LIN {X 0,Y 460.515,Z 491.122,A -85,B 0,C 180,E1 -7852.428,E2 -7852.428} C_VEL
LIN {X 0,Y 460.552,Z 491.116,A -85,B 0,C 180,E1 -7855.796,E2 -7855.796} C_VEL
LIN {X 0,Y 460.531,Z 491.12,A -85,B 0,C 180,E1 -7858.234,E2 -7858.234} C_VEL
LIN {X 0,Y 460.525,Z 491.123,A -85,B 0,C 180,E1 -7861.283,E2 -7861.283} C_VEL
LIN {X 0,Y 460.526,Z 491.122,A -85,B 0,C 180,E1 -7864.503,E2 -7864.503} C_VEL
LIN {X 0,Y 460.502,Z 491.122,A -85,B 0,C 180,E1 -7867.623,E2 -7867.623} C_VEL
LIN {X 0,Y 460.528,Z 491.12,A -85,B 0,C 180,E1 -7870.267,E2 -7870.267} C_VEL
LIN {X 0,Y 460.507,Z 491.124,A -85,B 0,C 180,E1 -7873.375,E2 -7873.375} C_VEL
LIN {X 0,Y 460.512,Z 491.123,A -85,B 0,C 180,E1 -7876.625,E2 -7876.625} C_VEL
LIN {X 0,Y 460.538,Z 491.117,A -85,B 0,C 180,E1 -7879.731,E2 -7879.731} C_VEL
LIN {X 0,Y 460.499,Z 491.125,A -85,B 0,C 180,E1 -7882.524,E2 -7882.524} C_VEL
LIN {X 0,Y 460.549,Z 491.116,A -85,B 0,C 180,E1 -7885.623,E2 -7885.623} C_VEL
LIN {X 0,Y 460.541,Z 491.119,A -85,B 0,C 180,E1 -7888.744,E2 -7888.744} C_VEL
LIN {X 0,Y 460.581,Z 491.112,A -85,B 0,C 180,E1 -7892.254,E2 -7892.254} C_VEL
LIN {X 0,Y 460.529,Z 491.12,A -85,B 0,C 180,E1 -7895.667,E2 -7895.667} C_VEL
LIN {X 0,Y 460.525,Z 491.121,A -85,B 0,C 180,E1 -7898.578,E2 -7898.578} C_VEL
LIN {X 0,Y 460.588,Z 491.114,A -85,B 0,C 180,E1 -7901.31,E2 -7901.31} C_VEL
LIN {X 0,Y 460.607,Z 491.108,A -85,B 0,C 180,E1 -7904.059,E2 -7904.059} C_VEL
LIN {X 0,Y 460.612,Z 491.11,A -85,B 0,C 180,E1 -7907.666,E2 -7907.666} C_VEL
LIN {X 0,Y 460.621,Z 491.108,A -85,B 0,C 180,E1 -7911.223,E2 -7911.223} C_VEL
LIN {X 0,Y 460.685,Z 491.1,A -85,B 0,C 180,E1 -7913.869,E2 -7913.869} C_VEL
LIN {X 0,Y 460.795,Z 491.086,A -85,B 0,C 180,E1 -7917.377,E2 -7917.377} C_VEL
LIN {X 0,Y 460.853,Z 491.079,A -85,B 0,C 180,E1 -7920,E2 -7920} C_VEL
LIN {X 0,Y 460.79,Z 491.09,A -85,B 0,C 180,E1 -7922.622,E2 -7922.622} C_VEL
LIN {X 0,Y 460.681,Z 491.101,A -85,B 0,C 180,E1 -7926.13,E2 -7926.13} C_VEL
LIN {X 0,Y 460.629,Z 491.11,A -85,B 0,C 180,E1 -7928.776,E2 -7928.776} C_VEL
LIN {X 0,Y 460.637,Z 491.106,A -85,B 0,C 180,E1 -7932.457,E2 -7932.457} C_VEL
LIN {X 0,Y 460.602,Z 491.111,A -85,B 0,C 180,E1 -7935.997,E2 -7935.997} C_VEL
LIN {X 0,Y 460.57,Z 491.112,A -85,B 0,C 180,E1 -7939.615,E2 -7939.615} C_VEL
LIN {X 0,Y 460.512,Z 491.123,A -85,B 0,C 180,E1 -7942.428,E2 -7942.428} C_VEL
LIN {X 0,Y 460.55,Z 491.115,A -85,B 0,C 180,E1 -7945.797,E2 -7945.797} C_VEL
LIN {X 0,Y 460.528,Z 491.122,A -85,B 0,C 180,E1 -7948.235,E2 -7948.235} C_VEL
LIN {X 0,Y 460.522,Z 491.12,A -85,B 0,C 180,E1 -7951.283,E2 -7951.283} C_VEL
LIN {X 0,Y 460.524,Z 491.121,A -85,B 0,C 180,E1 -7954.504,E2 -7954.504} C_VEL
LIN {X 0,Y 460.502,Z 491.121,A -85,B 0,C 180,E1 -7957.623,E2 -7957.623} C_VEL
LIN {X 0,Y 460.54,Z 491.121,A -85,B 0,C 180,E1 -7960.269,E2 -7960.269} C_VEL
LIN {X 0,Y 460.5,Z 491.123,A -85,B 0,C 180,E1 -7963.375,E2 -7963.375} C_VEL
LIN {X 0,Y 460.509,Z 491.118,A -85,B 0,C 180,E1 -7966.626,E2 -7966.626} C_VEL
LIN {X 0,Y 460.567,Z 491.21,A -85,B 0,C 180,E1 -7968.772,E2 -7968.772} C_VEL
LIN {X 0,Y 462.857,Z 502.692,A -85,B 0,C 180,E1 -7972.145,E2 -7972.145} C_VEL
LIN {X 0,Y 463.542,Z 507.45,A -85,B 0,C 180,E1 -7973.472,E2 -7973.472} C_VEL
LIN {X 0,Y 463.077,Z 516.53,A -85,B 0,C 180,E1 -7975.838,E2 -7975.838} C_VEL
LIN {X 0,Y 462.397,Z 530.597,A -85,B 0,C 180,E1 -7979.391,E2 -7979.391} C_VEL
LIN {X 0,Y 461.742,Z 544.673,A -85,B 0,C 180,E1 -7982.831,E2 -7982.831} C_VEL
LIN {X 0,Y 461.237,Z 558.404,A -85,B 0,C 180,E1 -7986.098,E2 -7986.098} C_VEL
LIN {X 0,Y 460.751,Z 572.777,A -85,B 0,C 180,E1 -7989.462,E2 -7989.462} C_VEL
LIN {X 0,Y 460.448,Z 586.76,A -85,B 0,C 180,E1 -7992.684,E2 -7992.684} C_VEL
LIN {X 0,Y 460.229,Z 593.953,A -85,B 0,C 180,E1 -7994.329,E2 -7994.329} C_VEL
LIN {X 0,Y 461.606,Z 608.371,A -85,B 0,C 180,E1 -7994.74,E2 -7994.74} C_VEL
LIN {X 0,Y 462.776,Z 619.695,A -85,B 0,C 180,E1 -7995.207,E2 -7995.207} C_VEL
LIN {X 0,Y 462.309,Z 631.594,A -85,B 0,C 180,E1 -7995.81,E2 -7995.81} C_VEL
LIN {X 0,Y 461.747,Z 643.169,A -85,B 0,C 180,E1 -7996.579,E2 -7996.579} C_VEL
LIN {X 0,Y 461.287,Z 654.794,A -85,B 0,C 180,E1 -7997.56,E2 -7997.56} C_VEL
LIN {X 0,Y 460.793,Z 664.432,A -85,B 0,C 180,E1 -7998.564,E2 -7998.564} C_VEL
LIN {X 0,Y 460.421,Z 673.14,A -85,B 0,C 180,E1 -7999.668,E2 -7999.668} C_VEL
LIN {X 0,Y 460.119,Z 681.62,A -85,B 0,C 180,E1 -8000.993,E2 -8000.993} C_VEL
LIN {X 0,Y 459.968,Z 688.469,A -85,B 0,C 180,E1 -8002.317,E2 -8002.317} C_VEL
LIN {X 0,Y 459.902,Z 694.757,A -85,B 0,C 180,E1 -8003.859,E2 -8003.859} C_VEL
LIN {X 0,Y 459.871,Z 698.831,A -85,B 0,C 180,E1 -8005.178,E2 -8005.178} C_VEL
LIN {X 0,Y 459.881,Z 701.832,A -85,B 0,C 180,E1 -8006.495,E2 -8006.495} C_VEL
LIN {X 0,Y 459.866,Z 703.258,A -85,B 0,C 180,E1 -8007.372,E2 -8007.372} C_VEL
LIN {X 0,Y 459.859,Z 704.259,A -85,B 0,C 180,E1 -8008.249,E2 -8008.249} C_VEL
LIN {X 0,Y 459.967,Z 705.067,A -85,B 0,C 180,E1 -8010,E2 -8010} C_VEL
LIN {X 0,Y 459.876,Z 704.13,A -85,B 0,C 180,E1 -8011.752,E2 -8011.752} C_VEL
LIN {X 0,Y 459.89,Z 703.058,A -85,B 0,C 180,E1 -8012.628,E2 -8012.628} C_VEL
LIN {X 0,Y 459.899,Z 701.567,A -85,B 0,C 180,E1 -8013.505,E2 -8013.505} C_VEL
LIN {X 0,Y 459.901,Z 698.452,A -85,B 0,C 180,E1 -8014.821,E2 -8014.821} C_VEL
LIN {X 0,Y 459.942,Z 694.259,A -85,B 0,C 180,E1 -8016.14,E2 -8016.14} C_VEL
LIN {X 0,Y 460.005,Z 687.828,A -85,B 0,C 180,E1 -8017.683,E2 -8017.683} C_VEL
LIN {X 0,Y 460.135,Z 680.836,A -85,B 0,C 180,E1 -8019.007,E2 -8019.007} C_VEL
LIN {X 0,Y 460.422,Z 672.202,A -85,B 0,C 180,E1 -8020.332,E2 -8020.332} C_VEL
LIN {X 0,Y 460.758,Z 662.35,A -85,B 0,C 180,E1 -8021.549,E2 -8021.549} C_VEL
LIN {X 0,Y 461.262,Z 652.412,A -85,B 0,C 180,E1 -8022.55,E2 -8022.55} C_VEL
LIN {X 0,Y 461.749,Z 641.834,A -85,B 0,C 180,E1 -8023.422,E2 -8023.422} C_VEL
LIN {X 0,Y 462.281,Z 630.154,A -85,B 0,C 180,E1 -8024.191,E2 -8024.191} C_VEL
LIN {X 0,Y 462.645,Z 618.154,A -85,B 0,C 180,E1 -8024.797,E2 -8024.797} C_VEL
LIN {X 0,Y 461.586,Z 608.526,A -85,B 0,C 180,E1 -8025.208,E2 -8025.208} C_VEL
LIN {X 0,Y 460.517,Z 595.101,A -85,B 0,C 180,E1 -8025.606,E2 -8025.606} C_VEL
LIN {X 0,Y 460.253,Z 591.872,A -85,B 0,C 180,E1 -8025.698,E2 -8025.698} C_VEL
LIN {X 0,Y 460.473,Z 578.368,A -85,B 0,C 180,E1 -8028.694,E2 -8028.694} C_VEL
LIN {X 0,Y 460.805,Z 562.857,A -85,B 0,C 180,E1 -8032.178,E2 -8032.178} C_VEL
LIN {X 0,Y 461.17,Z 547.892,A -85,B 0,C 180,E1 -8035.613,E2 -8035.613} C_VEL
LIN {X 0,Y 461.528,Z 534.973,A -85,B 0,C 180,E1 -8038.664,E2 -8038.664} C_VEL
LIN {X 0,Y 462.035,Z 522.031,A -85,B 0,C 180,E1 -8041.828,E2 -8041.828} C_VEL
LIN {X 0,Y 462.623,Z 508.615,A -85,B 0,C 180,E1 -8045.26,E2 -8045.26} C_VEL
LIN {X 0,Y 462.872,Z 504.269,A -85,B 0,C 180,E1 -8046.416,E2 -8046.416} C_VEL
LIN {X 0,Y 461.961,Z 498.32,A -85,B 0,C 180,E1 -8048.127,E2 -8048.127} C_VEL
LIN {X 0,Y 460.573,Z 491.117,A -85,B 0,C 180,E1 -8050.35,E2 -8050.35} C_VEL
LIN {X 0,Y 460.503,Z 491.127,A -85,B 0,C 180,E1 -8053.376,E2 -8053.376} C_VEL
LIN {X 0,Y 460.503,Z 491.127,A -85,B 0,C 180,E1 -8056.625,E2 -8056.625} C_VEL
LIN {X 0,Y 460.545,Z 491.121,A -85,B 0,C 180,E1 -8059.731,E2 -8059.731} C_VEL
LIN {X 0,Y 460.5,Z 491.127,A -85,B 0,C 180,E1 -8062.525,E2 -8062.525} C_VEL
LIN {X 0,Y 460.539,Z 491.118,A -85,B 0,C 180,E1 -8065.623,E2 -8065.623} C_VEL
LIN {X 0,Y 460.54,Z 491.119,A -85,B 0,C 180,E1 -8068.745,E2 -8068.745} C_VEL
LIN {X 0,Y 460.585,Z 491.115,A -85,B 0,C 180,E1 -8072.254,E2 -8072.254} C_VEL
LIN {X 0,Y 460.543,Z 491.119,A -85,B 0,C 180,E1 -8074.705,E2 -8074.705} C_VEL
LIN {X 0,Y 460.514,Z 491.122,A -85,B 0,C 180,E1 -8077.572,E2 -8077.572} C_VEL
LIN {X 0,Y 460.572,Z 491.115,A -85,B 0,C 180,E1 -8080.385,E2 -8080.385} C_VEL
LIN {X 0,Y 460.608,Z 491.111,A -85,B 0,C 180,E1 -8084.059,E2 -8084.059} C_VEL
LIN {X 0,Y 460.613,Z 491.109,A -85,B 0,C 180,E1 -8087.666,E2 -8087.666} C_VEL
LIN {X 0,Y 460.631,Z 491.106,A -85,B 0,C 180,E1 -8091.224,E2 -8091.224} C_VEL
LIN {X 0,Y 460.714,Z 491.098,A -85,B 0,C 180,E1 -8093.87,E2 -8093.87} C_VEL
LIN {X 0,Y 460.793,Z 491.089,A -85,B 0,C 180,E1 -8097.378,E2 -8097.378} C_VEL
LIN {X 0,Y 460.856,Z 491.08,A -85,B 0,C 180,E1 -8100,E2 -8100} C_VEL
LIN {X 0,Y 460.804,Z 491.087,A -85,B 0,C 180,E1 -8102.623,E2 -8102.623} C_VEL
LIN {X 0,Y 460.684,Z 491.099,A -85,B 0,C 180,E1 -8106.131,E2 -8106.131} C_VEL
LIN {X 0,Y 460.632,Z 491.106,A -85,B 0,C 180,E1 -8108.776,E2 -8108.776} C_VEL
LIN {X 0,Y 460.618,Z 491.111,A -85,B 0,C 180,E1 -8112.445,E2 -8112.445} C_VEL
LIN {X 0,Y 460.605,Z 491.114,A -85,B 0,C 180,E1 -8115.998,E2 -8115.998} C_VEL
LIN {X 0,Y 460.6,Z 491.118,A -85,B 0,C 180,E1 -8119.2,E2 -8119.2} C_VEL
LIN {X 0,Y 463.456,Z 501.008,A -85,B 0,C 180,E1 -8119.852,E2 -8119.852} C_VEL
LIN {X 0,Y 463.213,Z 512.77,A -85,B 0,C 180,E1 -8120.656,E2 -8120.656} C_VEL
LIN {X 0,Y 462.751,Z 523.16,A -85,B 0,C 180,E1 -8121.552,E2 -8121.552} C_VEL
LIN {X 0,Y 462.211,Z 533.805,A -85,B 0,C 180,E1 -8122.696,E2 -8122.696} C_VEL
LIN {X 0,Y 461.756,Z 542.796,A -85,B 0,C 180,E1 -8123.913,E2 -8123.913} C_VEL
LIN {X 0,Y 461.299,Z 550.763,A -85,B 0,C 180,E1 -8125.252,E2 -8125.252} C_VEL
LIN {X 0,Y 460.951,Z 557.693,A -85,B 0,C 180,E1 -8126.73,E2 -8126.73} C_VEL
LIN {X 0,Y 460.645,Z 563.061,A -85,B 0,C 180,E1 -8128.227,E2 -8128.227} C_VEL
LIN {X 0,Y 460.477,Z 566.619,A -85,B 0,C 180,E1 -8129.545,E2 -8129.545} C_VEL
LIN {X 0,Y 460.281,Z 569.813,A -85,B 0,C 180,E1 -8131.275,E2 -8131.275} C_VEL
LIN {X 0,Y 460.157,Z 571.303,A -85,B 0,C 180,E1 -8132.857,E2 -8132.857} C_VEL
LIN {X 0,Y 460.129,Z 571.523,A -85,B 0,C 180,E1 -8134.432,E2 -8134.432} C_VEL
LIN {X 0,Y 460.139,Z 570.552,A -85,B 0,C 180,E1 -8135.952,E2 -8135.952} C_VEL
LIN {X 0,Y 460.265,Z 568.06,A -85,B 0,C 180,E1 -8137.646,E2 -8137.646} C_VEL
LIN {X 0,Y 460.451,Z 564.012,A -85,B 0,C 180,E1 -8139.326,E2 -8139.326} C_VEL
LIN {X 0,Y 460.647,Z 559.848,A -85,B 0,C 180,E1 -8140.59,E2 -8140.59} C_VEL
LIN {X 0,Y 460.947,Z 553.302,A -85,B 0,C 180,E1 -8142.134,E2 -8142.134} C_VEL
LIN {X 0,Y 461.37,Z 545.39,A -85,B 0,C 180,E1 -8143.575,E2 -8143.575} C_VEL
LIN {X 0,Y 461.841,Z 536.372,A -85,B 0,C 180,E1 -8144.887,E2 -8144.887} C_VEL
LIN {X 0,Y 462.317,Z 526.16,A -85,B 0,C 180,E1 -8146.07,E2 -8146.07} C_VEL
LIN {X 0,Y 462.788,Z 514.9,A -85,B 0,C 180,E1 -8147.116,E2 -8147.116} C_VEL
LIN {X 0,Y 463.232,Z 503.54,A -85,B 0,C 180,E1 -8147.942,E2 -8147.942} C_VEL
LIN {X 0,Y 463.212,Z 500.817,A -85,B 0,C 180,E1 -8148.119,E2 -8148.119} C_VEL
LIN {X 0,Y 460.546,Z 491.136,A -85,B 0,C 180,E1 -8148.756,E2 -8148.756} C_VEL
LIN {X 0,Y 460.52,Z 491.123,A -85,B 0,C 180,E1 -8151.266,E2 -8151.266} C_VEL
LIN {X 0,Y 460.514,Z 491.121,A -85,B 0,C 180,E1 -8154.554,E2 -8154.554} C_VEL
LIN {X 0,Y 460.537,Z 491.119,A -85,B 0,C 180,E1 -8157.716,E2 -8157.716} C_VEL
LIN {X 0,Y 460.543,Z 491.117,A -85,B 0,C 180,E1 -8160.769,E2 -8160.769} C_VEL
LIN {X 0,Y 460.548,Z 491.118,A -85,B 0,C 180,E1 -8163.734,E2 -8163.734} C_VEL
LIN {X 0,Y 460.549,Z 491.116,A -85,B 0,C 180,E1 -8166.624,E2 -8166.624} C_VEL
LIN {X 0,Y 460.556,Z 491.117,A -85,B 0,C 180,E1 -8169.453,E2 -8169.453} C_VEL
LIN {X 0,Y 460.553,Z 491.116,A -85,B 0,C 180,E1 -8172.23,E2 -8172.23} C_VEL
LIN {X 0,Y 460.543,Z 491.116,A -85,B 0,C 180,E1 -8172.589,E2 -8172.589} C_VEL
LIN {X 0,Y 459.876,Z 491.204,A -85,B 0,C 180,E1 -8173.319,E2 -8173.319} C_VEL
LIN {X 0,Y 457.008,Z 491.557,A -85,B 0,C 180,E1 -8174.504,E2 -8174.504} C_VEL
LIN {X 0,Y 454.594,Z 491.86,A -85,B 0,C 180,E1 -8175.461,E2 -8175.461} C_VEL
LIN {X 0,Y 453.576,Z 491.986,A -85,B 0,C 180,E1 -8176.2,E2 -8176.2} C_VEL
LIN {X 0,Y 453.504,Z 491.995,A -85,B 0,C 180,E1 -8176.45,E2 -8176.45} C_VEL
LIN {X 0,Y 453.536,Z 491.993,A -85,B 0,C 180,E1 -8179.283,E2 -8179.283} C_VEL
LIN {X 0,Y 453.636,Z 491.979,A -85,B 0,C 180,E1 -8182.54,E2 -8182.54} C_VEL
LIN {X 0,Y 453.663,Z 491.974,A -85,B 0,C 180,E1 -8184.667,E2 -8184.667} C_VEL
LIN {X 0,Y 453.75,Z 491.965,A -85,B 0,C 180,E1 -8187.337,E2 -8187.337} C_VEL
LIN {X 0,Y 453.821,Z 491.955,A -85,B 0,C 180,E1 -8190,E2 -8190} C_VEL
LIN {X 0,Y 453.741,Z 491.965,A -85,B 0,C 180,E1 -8192.663,E2 -8192.663} C_VEL
LIN {X 0,Y 453.649,Z 491.976,A -85,B 0,C 180,E1 -8196.226,E2 -8196.226} C_VEL
LIN {X 0,Y 453.591,Z 491.986,A -85,B 0,C 180,E1 -8198.913,E2 -8198.913} C_VEL
LIN {X 0,Y 453.569,Z 491.986,A -85,B 0,C 180,E1 -8202.529,E2 -8202.529} C_VEL
LIN {X 0,Y 453.549,Z 491.989,A -85,B 0,C 180,E1 -8206.196,E2 -8206.196} C_VEL
LIN {X 0,Y 453.522,Z 491.994,A -85,B 0,C 180,E1 -8209.039,E2 -8209.039} C_VEL
LIN {X 0,Y 453.481,Z 491.999,A -85,B 0,C 180,E1 -8211.836,E2 -8211.836} C_VEL
LIN {X 0,Y 453.499,Z 491.995,A -85,B 0,C 180,E1 -8214.735,E2 -8214.735} C_VEL
LIN {X 0,Y 453.511,Z 491.994,A -85,B 0,C 180,E1 -8217.953,E2 -8217.953} C_VEL
LIN {X 0,Y 453.479,Z 491.998,A -85,B 0,C 180,E1 -8220.759,E2 -8220.759} C_VEL
LIN {X 0,Y 453.472,Z 491.999,A -85,B 0,C 180,E1 -8223.913,E2 -8223.913} C_VEL
LIN {X 0,Y 453.453,Z 492.005,A -85,B 0,C 180,E1 -8227.19,E2 -8227.19} C_VEL
LIN {X 0,Y 453.474,Z 492,A -85,B 0,C 180,E1 -8230.611,E2 -8230.611} C_VEL
LIN {X 0,Y 453.463,Z 491.998,A -85,B 0,C 180,E1 -8234.222,E2 -8234.222} C_VEL
LIN {X 0,Y 453.451,Z 492.002,A -85,B 0,C 180,E1 -8237.003,E2 -8237.003} C_VEL
LIN {X 0,Y 453.497,Z 491.996,A -85,B 0,C 180,E1 -8239.409,E2 -8239.409} C_VEL
LIN {X 0,Y 453.452,Z 492.002,A -85,B 0,C 180,E1 -8242.81,E2 -8242.81} C_VEL
LIN {X 0,Y 453.48,Z 491.996,A -85,B 0,C 180,E1 -8246.087,E2 -8246.087} C_VEL
LIN {X 0,Y 453.48,Z 491.999,A -85,B 0,C 180,E1 -8249.24,E2 -8249.24} C_VEL
LIN {X 0,Y 453.536,Z 491.989,A -85,B 0,C 180,E1 -8252.297,E2 -8252.297} C_VEL
LIN {X 0,Y 453.499,Z 491.997,A -85,B 0,C 180,E1 -8255.264,E2 -8255.264} C_VEL
LIN {X 0,Y 453.483,Z 491.997,A -85,B 0,C 180,E1 -8258.415,E2 -8258.415} C_VEL
LIN {X 0,Y 453.525,Z 491.993,A -85,B 0,C 180,E1 -8261.008,E2 -8261.008} C_VEL
LIN {X 0,Y 453.572,Z 491.984,A -85,B 0,C 180,E1 -8263.879,E2 -8263.879} C_VEL
LIN {X 0,Y 453.567,Z 491.989,A -85,B 0,C 180,E1 -8267.471,E2 -8267.471} C_VEL
LIN {X 0,Y 453.587,Z 491.985,A -85,B 0,C 180,E1 -8271.086,E2 -8271.086} C_VEL
LIN {X 0,Y 453.651,Z 491.976,A -85,B 0,C 180,E1 -8273.774,E2 -8273.774} C_VEL
LIN {X 0,Y 453.739,Z 491.965,A -85,B 0,C 180,E1 -8277.336,E2 -8277.336} C_VEL
LIN {X 0,Y 453.822,Z 491.955,A -85,B 0,C 180,E1 -8280,E2 -8280} C_VEL
LIN {X 0,Y 453.733,Z 491.969,A -85,B 0,C 180,E1 -8282.663,E2 -8282.663} C_VEL
LIN {X 0,Y 453.648,Z 491.977,A -85,B 0,C 180,E1 -8286.226,E2 -8286.226} C_VEL
LIN {X 0,Y 453.593,Z 491.985,A -85,B 0,C 180,E1 -8288.913,E2 -8288.913} C_VEL
LIN {X 0,Y 453.604,Z 491.982,A -85,B 0,C 180,E1 -8292.55,E2 -8292.55} C_VEL
LIN {X 0,Y 453.546,Z 491.991,A -85,B 0,C 180,E1 -8296.196,E2 -8296.196} C_VEL
LIN {X 0,Y 453.52,Z 491.995,A -85,B 0,C 180,E1 -8299.039,E2 -8299.039} C_VEL
LIN {X 0,Y 453.478,Z 491.998,A -85,B 0,C 180,E1 -8301.836,E2 -8301.836} C_VEL
LIN {X 0,Y 453.501,Z 491.997,A -85,B 0,C 180,E1 -8304.735,E2 -8304.735} C_VEL
LIN {X 0,Y 453.492,Z 491.996,A -85,B 0,C 180,E1 -8307.949,E2 -8307.949} C_VEL
LIN {X 0,Y 453.477,Z 492,A -85,B 0,C 180,E1 -8310.759,E2 -8310.759} C_VEL
LIN {X 0,Y 453.469,Z 491.999,A -85,B 0,C 180,E1 -8313.913,E2 -8313.913} C_VEL
LIN {X 0,Y 453.453,Z 492.001,A -85,B 0,C 180,E1 -8317.19,E2 -8317.19} C_VEL
LIN {X 0,Y 453.495,Z 491.997,A -85,B 0,C 180,E1 -8320.609,E2 -8320.609} C_VEL
LIN {X 0,Y 453.456,Z 492.001,A -85,B 0,C 180,E1 -8323.244,E2 -8323.244} C_VEL
LIN {X 0,Y 453.461,Z 491.998,A -85,B 0,C 180,E1 -8325.778,E2 -8325.778} C_VEL
LIN {X 0,Y 453.487,Z 492.004,A -85,B 0,C 180,E1 -8328.445,E2 -8328.445} C_VEL
LIN {X 0,Y 455.388,Z 501.552,A -85,B 0,C 180,E1 -8331.316,E2 -8331.316} C_VEL
LIN {X 0,Y 456.563,Z 507.989,A -85,B 0,C 180,E1 -8333.173,E2 -8333.173} C_VEL
LIN {X 0,Y 456.325,Z 514.75,A -85,B 0,C 180,E1 -8334.979,E2 -8334.979} C_VEL
LIN {X 0,Y 455.536,Z 528.839,A -85,B 0,C 180,E1 -8338.621,E2 -8338.621} C_VEL
LIN {X 0,Y 454.948,Z 539.861,A -85,B 0,C 180,E1 -8341.387,E2 -8341.387} C_VEL
LIN {X 0,Y 454.38,Z 553.898,A -85,B 0,C 180,E1 -8344.827,E2 -8344.827} C_VEL
LIN {X 0,Y 453.842,Z 567.913,A -85,B 0,C 180,E1 -8348.182,E2 -8348.182} C_VEL
LIN {X 0,Y 453.505,Z 579.893,A -85,B 0,C 180,E1 -8351.008,E2 -8351.008} C_VEL
LIN {X 0,Y 453.186,Z 593.062,A -85,B 0,C 180,E1 -8354.084,E2 -8354.084} C_VEL
LIN {X 0,Y 454.691,Z 608.653,A -85,B 0,C 180,E1 -8354.55,E2 -8354.55} C_VEL
LIN {X 0,Y 455.77,Z 621.036,A -85,B 0,C 180,E1 -8355.089,E2 -8355.089} C_VEL
LIN {X 0,Y 455.205,Z 634.072,A -85,B 0,C 180,E1 -8355.812,E2 -8355.812} C_VEL
LIN {X 0,Y 454.66,Z 644.956,A -85,B 0,C 180,E1 -8356.593,E2 -8356.593} C_VEL
LIN {X 0,Y 454.238,Z 655.045,A -85,B 0,C 180,E1 -8357.49,E2 -8357.49} C_VEL
LIN {X 0,Y 453.708,Z 665.245,A -85,B 0,C 180,E1 -8358.609,E2 -8358.609} C_VEL
LIN {X 0,Y 453.229,Z 675.123,A -85,B 0,C 180,E1 -8359.954,E2 -8359.954} C_VEL
LIN {X 0,Y 453.003,Z 683.058,A -85,B 0,C 180,E1 -8361.3,E2 -8361.3} C_VEL
LIN {X 0,Y 452.867,Z 688.468,A -85,B 0,C 180,E1 -8362.42,E2 -8362.42} C_VEL
LIN {X 0,Y 452.825,Z 693.739,A -85,B 0,C 180,E1 -8363.763,E2 -8363.763} C_VEL
LIN {X 0,Y 452.825,Z 697.82,A -85,B 0,C 180,E1 -8365.103,E2 -8365.103} C_VEL
LIN {X 0,Y 452.839,Z 700.822,A -85,B 0,C 180,E1 -8366.441,E2 -8366.441} C_VEL
LIN {X 0,Y 452.824,Z 702.247,A -85,B 0,C 180,E1 -8367.331,E2 -8367.331} C_VEL
LIN {X 0,Y 452.824,Z 703.248,A -85,B 0,C 180,E1 -8368.221,E2 -8368.221} C_VEL
LIN {X 0,Y 452.952,Z 704.052,A -85,B 0,C 180,E1 -8370,E2 -8370} C_VEL
LIN {X 0,Y 452.843,Z 703.103,A -85,B 0,C 180,E1 -8371.779,E2 -8371.779} C_VEL
LIN {X 0,Y 452.85,Z 702.026,A -85,B 0,C 180,E1 -8372.669,E2 -8372.669} C_VEL
LIN {X 0,Y 452.857,Z 700.526,A -85,B 0,C 180,E1 -8373.559,E2 -8373.559} C_VEL
LIN {X 0,Y 452.86,Z 697.4,A -85,B 0,C 180,E1 -8374.897,E2 -8374.897} C_VEL
LIN {X 0,Y 452.888,Z 693.193,A -85,B 0,C 180,E1 -8376.236,E2 -8376.236} C_VEL
LIN {X 0,Y 452.925,Z 686.743,A -85,B 0,C 180,E1 -8377.803,E2 -8377.803} C_VEL
LIN {X 0,Y 453.088,Z 679.737,A -85,B 0,C 180,E1 -8379.149,E2 -8379.149} C_VEL
LIN {X 0,Y 453.369,Z 671.082,A -85,B 0,C 180,E1 -8380.495,E2 -8380.495} C_VEL
LIN {X 0,Y 453.676,Z 662.218,A -85,B 0,C 180,E1 -8381.618,E2 -8381.618} C_VEL
LIN {X 0,Y 454.196,Z 652.578,A -85,B 0,C 180,E1 -8382.624,E2 -8382.624} C_VEL
LIN {X 0,Y 454.788,Z 640.678,A -85,B 0,C 180,E1 -8383.631,E2 -8383.631} C_VEL
LIN {X 0,Y 455.36,Z 629.001,A -85,B 0,C 180,E1 -8384.411,E2 -8384.411} C_VEL
LIN {X 0,Y 455.64,Z 618.328,A -85,B 0,C 180,E1 -8384.973,E2 -8384.973} C_VEL
LIN {X 0,Y 454.677,Z 609.071,A -85,B 0,C 180,E1 -8385.386,E2 -8385.386} C_VEL
LIN {X 0,Y 453.648,Z 595.57,A -85,B 0,C 180,E1 -8385.825,E2 -8385.825} C_VEL
LIN {X 0,Y 453.159,Z 590.712,A -85,B 0,C 180,E1 -8385.955,E2 -8385.955} C_VEL
LIN {X 0,Y 453.429,Z 577.222,A -85,B 0,C 180,E1 -8389.006,E2 -8389.006} C_VEL
LIN {X 0,Y 453.732,Z 561.811,A -85,B 0,C 180,E1 -8392.542,E2 -8392.542} C_VEL
LIN {X 0,Y 454.164,Z 547.39,A -85,B 0,C 180,E1 -8395.926,E2 -8395.926} C_VEL
LIN {X 0,Y 454.564,Z 534.06,A -85,B 0,C 180,E1 -8399.145,E2 -8399.145} C_VEL
LIN {X 0,Y 455.081,Z 521.732,A -85,B 0,C 180,E1 -8402.232,E2 -8402.232} C_VEL
LIN {X 0,Y 455.709,Z 509.384,A -85,B 0,C 180,E1 -8405.466,E2 -8405.466} C_VEL
LIN {X 0,Y 455.881,Z 504.829,A -85,B 0,C 180,E1 -8406.712,E2 -8406.712} C_VEL
LIN {X 0,Y 454.315,Z 496.021,A -85,B 0,C 180,E1 -8409.365,E2 -8409.365} C_VEL
LIN {X 0,Y 453.517,Z 491.994,A -85,B 0,C 180,E1 -8410.68,E2 -8410.68} C_VEL
LIN {X 0,Y 453.469,Z 492.003,A -85,B 0,C 180,E1 -8414.221,E2 -8414.221} C_VEL
LIN {X 0,Y 453.466,Z 492.003,A -85,B 0,C 180,E1 -8417.005,E2 -8417.005} C_VEL
LIN {X 0,Y 453.497,Z 491.999,A -85,B 0,C 180,E1 -8419.409,E2 -8419.409} C_VEL
LIN {X 0,Y 453.45,Z 492.002,A -85,B 0,C 180,E1 -8422.228,E2 -8422.228} C_VEL
LIN {X 0,Y 453.484,Z 491.998,A -85,B 0,C 180,E1 -8425.224,E2 -8425.224} C_VEL
LIN {X 0,Y 453.469,Z 491.998,A -85,B 0,C 180,E1 -8428.475,E2 -8428.475} C_VEL
LIN {X 0,Y 453.536,Z 491.991,A -85,B 0,C 180,E1 -8432.041,E2 -8432.041} C_VEL
LIN {X 0,Y 453.504,Z 491.993,A -85,B 0,C 180,E1 -8435.265,E2 -8435.265} C_VEL
LIN {X 0,Y 453.484,Z 491.998,A -85,B 0,C 180,E1 -8438.415,E2 -8438.415} C_VEL
LIN {X 0,Y 453.526,Z 491.994,A -85,B 0,C 180,E1 -8441.009,E2 -8441.009} C_VEL
LIN {X 0,Y 453.573,Z 491.988,A -85,B 0,C 180,E1 -8443.88,E2 -8443.88} C_VEL
LIN {X 0,Y 453.568,Z 491.988,A -85,B 0,C 180,E1 -8447.471,E2 -8447.471} C_VEL
LIN {X 0,Y 453.595,Z 491.983,A -85,B 0,C 180,E1 -8451.087,E2 -8451.087} C_VEL
LIN {X 0,Y 453.682,Z 491.974,A -85,B 0,C 180,E1 -8453.775,E2 -8453.775} C_VEL
LIN {X 0,Y 453.736,Z 491.968,A -85,B 0,C 180,E1 -8457.337,E2 -8457.337} C_VEL
LIN {X 0,Y 453.826,Z 491.956,A -85,B 0,C 180,E1 -8460,E2 -8460} C_VEL
LIN {X 0,Y 453.748,Z 491.966,A -85,B 0,C 180,E1 -8462.664,E2 -8462.664} C_VEL
LIN {X 0,Y 453.65,Z 491.975,A -85,B 0,C 180,E1 -8466.226,E2 -8466.226} C_VEL
LIN {X 0,Y 453.596,Z 491.982,A -85,B 0,C 180,E1 -8468.914,E2 -8468.914} C_VEL
LIN {X 0,Y 453.568,Z 491.988,A -85,B 0,C 180,E1 -8472.529,E2 -8472.529} C_VEL
LIN {X 0,Y 453.549,Z 491.992,A -85,B 0,C 180,E1 -8476.196,E2 -8476.196} C_VEL
LIN {X 0,Y 453.582,Z 491.992,A -85,B 0,C 180,E1 -8478.938,E2 -8478.938} C_VEL
LIN {X 0,Y 456.704,Z 502.758,A -85,B 0,C 180,E1 -8479.672,E2 -8479.672} C_VEL
LIN {X 0,Y 456.378,Z 514.33,A -85,B 0,C 180,E1 -8480.485,E2 -8480.485} C_VEL
LIN {X 0,Y 455.861,Z 525.491,A -85,B 0,C 180,E1 -8481.479,E2 -8481.479} C_VEL
LIN {X 0,Y 455.348,Z 535.146,A -85,B 0,C 180,E1 -8482.549,E2 -8482.549} C_VEL
LIN {X 0,Y 454.894,Z 543.44,A -85,B 0,C 180,E1 -8483.684,E2 -8483.684} C_VEL
LIN {X 0,Y 454.434,Z 550.853,A -85,B 0,C 180,E1 -8484.925,E2 -8484.925} C_VEL
LIN {X 0,Y 454.084,Z 557.705,A -85,B 0,C 180,E1 -8486.359,E2 -8486.359} C_VEL
LIN {X 0,Y 453.748,Z 562.725,A -85,B 0,C 180,E1 -8487.689,E2 -8487.689} C_VEL
LIN {X 0,Y 453.524,Z 567.102,A -85,B 0,C 180,E1 -8489.219,E2 -8489.219} C_VEL
LIN {X 0,Y 453.309,Z 570.173,A -85,B 0,C 180,E1 -8490.773,E2 -8490.773} C_VEL
LIN {X 0,Y 453.224,Z 571.546,A -85,B 0,C 180,E1 -8491.819,E2 -8491.819} C_VEL
LIN {X 0,Y 453.149,Z 572.462,A -85,B 0,C 180,E1 -8493.122,E2 -8493.122} C_VEL
LIN {X 0,Y 453.118,Z 572.475,A -85,B 0,C 180,E1 -8494.709,E2 -8494.709} C_VEL
LIN {X 0,Y 453.145,Z 571.288,A -85,B 0,C 180,E1 -8496.245,E2 -8496.245} C_VEL
LIN {X 0,Y 453.252,Z 568.974,A -85,B 0,C 180,E1 -8497.74,E2 -8497.74} C_VEL
LIN {X 0,Y 453.469,Z 564.857,A -85,B 0,C 180,E1 -8499.452,E2 -8499.452} C_VEL
LIN {X 0,Y 453.767,Z 558.988,A -85,B 0,C 180,E1 -8501.166,E2 -8501.166} C_VEL
LIN {X 0,Y 454.083,Z 552.22,A -85,B 0,C 180,E1 -8502.663,E2 -8502.663} C_VEL
LIN {X 0,Y 454.501,Z 545.332,A -85,B 0,C 180,E1 -8503.88,E2 -8503.88} C_VEL
LIN {X 0,Y 454.955,Z 536.826,A -85,B 0,C 180,E1 -8505.107,E2 -8505.107} C_VEL
LIN {X 0,Y 455.378,Z 527.828,A -85,B 0,C 180,E1 -8506.168,E2 -8506.168} C_VEL
LIN {X 0,Y 455.857,Z 517.048,A -85,B 0,C 180,E1 -8507.2,E2 -8507.2} C_VEL
LIN {X 0,Y 456.328,Z 506.14,A -85,B 0,C 180,E1 -8508.034,E2 -8508.034} C_VEL
LIN {X 0,Y 456.398,Z 502.612,A -85,B 0,C 180,E1 -8508.264,E2 -8508.264} C_VEL
LIN {X 0,Y 453.497,Z 491.997,A -85,B 0,C 180,E1 -8508.988,E2 -8508.988} C_VEL
LIN {X 0,Y 453.451,Z 492.004,A -85,B 0,C 180,E1 -8512.228,E2 -8512.228} C_VEL
LIN {X 0,Y 453.492,Z 491.997,A -85,B 0,C 180,E1 -8515.223,E2 -8515.223} C_VEL
LIN {X 0,Y 453.471,Z 491.999,A -85,B 0,C 180,E1 -8518.475,E2 -8518.475} C_VEL
LIN {X 0,Y 453.534,Z 491.99,A -85,B 0,C 180,E1 -8522.041,E2 -8522.041} C_VEL
LIN {X 0,Y 453.501,Z 491.996,A -85,B 0,C 180,E1 -8525.265,E2 -8525.265} C_VEL
LIN {X 0,Y 453.486,Z 491.996,A -85,B 0,C 180,E1 -8528.415,E2 -8528.415} C_VEL
LIN {X 0,Y 453.528,Z 491.992,A -85,B 0,C 180,E1 -8531.009,E2 -8531.009} C_VEL
LIN {X 0,Y 453.575,Z 491.985,A -85,B 0,C 180,E1 -8533.88,E2 -8533.88} C_VEL
LIN {X 0,Y 453.504,Z 491.995,A -85,B 0,C 180,E1 -8536.45,E2 -8536.45} C_VEL
LIN {X 0,Y 452.869,Z 492.077,A -85,B 0,C 180,E1 -8537.191,E2 -8537.191} C_VEL
LIN {X 0,Y 450.04,Z 492.428,A -85,B 0,C 180,E1 -8538.396,E2 -8538.396} C_VEL
LIN {X 0,Y 447.632,Z 492.73,A -85,B 0,C 180,E1 -8539.368,E2 -8539.368} C_VEL
LIN {X 0,Y 446.6,Z 492.853,A -85,B 0,C 180,E1 -8540.118,E2 -8540.118} C_VEL
LIN {X 0,Y 446.518,Z 492.863,A -85,B 0,C 180,E1 -8540.373,E2 -8540.373} C_VEL
LIN {X 0,Y 446.618,Z 492.855,A -85,B 0,C 180,E1 -8543.676,E2 -8543.676} C_VEL
LIN {X 0,Y 446.697,Z 492.844,A -85,B 0,C 180,E1 -8547.295,E2 -8547.295} C_VEL
LIN {X 0,Y 446.79,Z 492.831,A -85,B 0,C 180,E1 -8550,E2 -8550} C_VEL
LIN {X 0,Y 446.688,Z 492.844,A -85,B 0,C 180,E1 -8552.705,E2 -8552.705} C_VEL
LIN {X 0,Y 446.617,Z 492.852,A -85,B 0,C 180,E1 -8556.324,E2 -8556.324} C_VEL
LIN {X 0,Y 446.538,Z 492.865,A -85,B 0,C 180,E1 -8559.055,E2 -8559.055} C_VEL
LIN {X 0,Y 446.527,Z 492.863,A -85,B 0,C 180,E1 -8562.73,E2 -8562.73} C_VEL
LIN {X 0,Y 446.501,Z 492.867,A -85,B 0,C 180,E1 -8566.227,E2 -8566.227} C_VEL
LIN {X 0,Y 446.473,Z 492.873,A -85,B 0,C 180,E1 -8569.303,E2 -8569.303} C_VEL
LIN {X 0,Y 446.423,Z 492.877,A -85,B 0,C 180,E1 -8572.199,E2 -8572.199} C_VEL
LIN {X 0,Y 446.443,Z 492.877,A -85,B 0,C 180,E1 -8575.153,E2 -8575.153} C_VEL
LIN {X 0,Y 446.453,Z 492.873,A -85,B 0,C 180,E1 -8578.181,E2 -8578.181} C_VEL
LIN {X 0,Y 446.42,Z 492.88,A -85,B 0,C 180,E1 -8581.3,E2 -8581.3} C_VEL
LIN {X 0,Y 446.426,Z 492.878,A -85,B 0,C 180,E1 -8584.523,E2 -8584.523} C_VEL
LIN {X 0,Y 446.414,Z 492.876,A -85,B 0,C 180,E1 -8588.078,E2 -8588.078} C_VEL
LIN {X 0,Y 446.41,Z 492.881,A -85,B 0,C 180,E1 -8591.393,E2 -8591.393} C_VEL
LIN {X 0,Y 446.453,Z 492.874,A -85,B 0,C 180,E1 -8595.104,E2 -8595.104} C_VEL
LIN {X 0,Y 446.422,Z 492.877,A -85,B 0,C 180,E1 -8598.608,E2 -8598.608} C_VEL
LIN {X 0,Y 446.427,Z 492.879,A -85,B 0,C 180,E1 -8600.971,E2 -8600.971} C_VEL
LIN {X 0,Y 446.42,Z 492.877,A -85,B 0,C 180,E1 -8604.373,E2 -8604.373} C_VEL
LIN {X 0,Y 446.426,Z 492.877,A -85,B 0,C 180,E1 -8607.638,E2 -8607.638} C_VEL
LIN {X 0,Y 446.452,Z 492.874,A -85,B 0,C 180,E1 -8610.79,E2 -8610.79} C_VEL
LIN {X 0,Y 446.463,Z 492.872,A -85,B 0,C 180,E1 -8613.847,E2 -8613.847} C_VEL
LIN {X 0,Y 446.428,Z 492.877,A -85,B 0,C 180,E1 -8616.823,E2 -8616.823} C_VEL
LIN {X 0,Y 446.446,Z 492.874,A -85,B 0,C 180,E1 -8619.737,E2 -8619.737} C_VEL
LIN {X 0,Y 446.459,Z 492.872,A -85,B 0,C 180,E1 -8622.597,E2 -8622.597} C_VEL
LIN {X 0,Y 446.471,Z 492.871,A -85,B 0,C 180,E1 -8625.412,E2 -8625.412} C_VEL
LIN {X 0,Y 446.52,Z 492.865,A -85,B 0,C 180,E1 -8628.193,E2 -8628.193} C_VEL
LIN {X 0,Y 446.535,Z 492.865,A -85,B 0,C 180,E1 -8630.944,E2 -8630.944} C_VEL
LIN {X 0,Y 446.619,Z 492.852,A -85,B 0,C 180,E1 -8633.676,E2 -8633.676} C_VEL
LIN {X 0,Y 446.686,Z 492.844,A -85,B 0,C 180,E1 -8637.294,E2 -8637.294} C_VEL
LIN {X 0,Y 446.792,Z 492.83,A -85,B 0,C 180,E1 -8640,E2 -8640} C_VEL
LIN {X 0,Y 446.68,Z 492.848,A -85,B 0,C 180,E1 -8642.705,E2 -8642.705} C_VEL
LIN {X 0,Y 446.617,Z 492.852,A -85,B 0,C 180,E1 -8646.324,E2 -8646.324} C_VEL
LIN {X 0,Y 446.539,Z 492.863,A -85,B 0,C 180,E1 -8649.055,E2 -8649.055} C_VEL
LIN {X 0,Y 446.536,Z 492.864,A -85,B 0,C 180,E1 -8652.729,E2 -8652.729} C_VEL
LIN {X 0,Y 446.49,Z 492.87,A -85,B 0,C 180,E1 -8656.459,E2 -8656.459} C_VEL
LIN {X 0,Y 446.47,Z 492.87,A -85,B 0,C 180,E1 -8659.303,E2 -8659.303} C_VEL
LIN {X 0,Y 446.42,Z 492.878,A -85,B 0,C 180,E1 -8662.199,E2 -8662.199} C_VEL
LIN {X 0,Y 446.444,Z 492.875,A -85,B 0,C 180,E1 -8665.153,E2 -8665.153} C_VEL
LIN {X 0,Y 446.441,Z 492.876,A -85,B 0,C 180,E1 -8668.182,E2 -8668.182} C_VEL
LIN {X 0,Y 446.417,Z 492.877,A -85,B 0,C 180,E1 -8671.3,E2 -8671.3} C_VEL
LIN {X 0,Y 446.424,Z 492.878,A -85,B 0,C 180,E1 -8674.523,E2 -8674.523} C_VEL
LIN {X 0,Y 446.414,Z 492.876,A -85,B 0,C 180,E1 -8678.079,E2 -8678.079} C_VEL
LIN {X 0,Y 446.429,Z 492.879,A -85,B 0,C 180,E1 -8681.391,E2 -8681.391} C_VEL
LIN {X 0,Y 446.452,Z 492.87,A -85,B 0,C 180,E1 -8685.104,E2 -8685.104} C_VEL
LIN {X 0,Y 446.45,Z 493.074,A -85,B 0,C 180,E1 -8688.193,E2 -8688.193} C_VEL
LIN {X 0,Y 448.423,Z 502.801,A -85,B 0,C 180,E1 -8691.178,E2 -8691.178} C_VEL
LIN {X 0,Y 449.653,Z 509.818,A -85,B 0,C 180,E1 -8693.229,E2 -8693.229} C_VEL
LIN {X 0,Y 449.159,Z 519.04,A -85,B 0,C 180,E1 -8695.716,E2 -8695.716} C_VEL
LIN {X 0,Y 448.412,Z 532.605,A -85,B 0,C 180,E1 -8699.258,E2 -8699.258} C_VEL
LIN {X 0,Y 447.637,Z 547.054,A -85,B 0,C 180,E1 -8702.915,E2 -8702.915} C_VEL
LIN {X 0,Y 447.128,Z 559.077,A -85,B 0,C 180,E1 -8705.879,E2 -8705.879} C_VEL
LIN {X 0,Y 446.634,Z 573.009,A -85,B 0,C 180,E1 -8709.265,E2 -8709.265} C_VEL
LIN {X 0,Y 446.29,Z 586.929,A -85,B 0,C 180,E1 -8712.59,E2 -8712.59} C_VEL
LIN {X 0,Y 446.152,Z 592.452,A -85,B 0,C 180,E1 -8713.852,E2 -8713.852} C_VEL
LIN {X 0,Y 447.535,Z 606.314,A -85,B 0,C 180,E1 -8714.26,E2 -8714.26} C_VEL
LIN {X 0,Y 448.487,Z 617.342,A -85,B 0,C 180,E1 -8714.725,E2 -8714.725} C_VEL
LIN {X 0,Y 448.76,Z 622.157,A -85,B 0,C 180,E1 -8714.967,E2 -8714.967} C_VEL
LIN {X 0,Y 448.185,Z 634.73,A -85,B 0,C 180,E1 -8715.701,E2 -8715.701} C_VEL
LIN {X 0,Y 447.564,Z 646.199,A -85,B 0,C 180,E1 -8716.574,E2 -8716.574} C_VEL
LIN {X 0,Y 447.154,Z 656.18,A -85,B 0,C 180,E1 -8717.519,E2 -8717.519} C_VEL
LIN {X 0,Y 446.644,Z 664.188,A -85,B 0,C 180,E1 -8718.427,E2 -8718.427} C_VEL
LIN {X 0,Y 446.193,Z 674.08,A -85,B 0,C 180,E1 -8719.793,E2 -8719.793} C_VEL
LIN {X 0,Y 445.932,Z 682.025,A -85,B 0,C 180,E1 -8721.161,E2 -8721.161} C_VEL
LIN {X 0,Y 445.822,Z 687.442,A -85,B 0,C 180,E1 -8722.3,E2 -8722.3} C_VEL
LIN {X 0,Y 445.756,Z 692.716,A -85,B 0,C 180,E1 -8723.664,E2 -8723.664} C_VEL
LIN {X 0,Y 445.778,Z 696.805,A -85,B 0,C 180,E1 -8725.026,E2 -8725.026} C_VEL
LIN {X 0,Y 445.799,Z 699.808,A -85,B 0,C 180,E1 -8726.385,E2 -8726.385} C_VEL
LIN {X 0,Y 445.783,Z 701.235,A -85,B 0,C 180,E1 -8727.289,E2 -8727.289} C_VEL
LIN {X 0,Y 445.788,Z 702.236,A -85,B 0,C 180,E1 -8728.193,E2 -8728.193} C_VEL
LIN {X 0,Y 445.936,Z 703.036,A -85,B 0,C 180,E1 -8730,E2 -8730} C_VEL
LIN {X 0,Y 445.809,Z 702.079,A -85,B 0,C 180,E1 -8731.807,E2 -8731.807} C_VEL
LIN {X 0,Y 445.81,Z 700.991,A -85,B 0,C 180,E1 -8732.711,E2 -8732.711} C_VEL
LIN {X 0,Y 445.816,Z 699.486,A -85,B 0,C 180,E1 -8733.615,E2 -8733.615} C_VEL
LIN {X 0,Y 445.817,Z 696.349,A -85,B 0,C 180,E1 -8734.974,E2 -8734.974} C_VEL
LIN {X 0,Y 445.811,Z 692.123,A -85,B 0,C 180,E1 -8736.336,E2 -8736.336} C_VEL
LIN {X 0,Y 445.877,Z 685.66,A -85,B 0,C 180,E1 -8737.928,E2 -8737.928} C_VEL
LIN {X 0,Y 446.042,Z 678.634,A -85,B 0,C 180,E1 -8739.294,E2 -8739.294} C_VEL
LIN {X 0,Y 446.341,Z 669.965,A -85,B 0,C 180,E1 -8740.662,E2 -8740.662} C_VEL
LIN {X 0,Y 446.747,Z 660.103,A -85,B 0,C 180,E1 -8741.916,E2 -8741.916} C_VEL
LIN {X 0,Y 447.104,Z 651.607,A -85,B 0,C 180,E1 -8742.814,E2 -8742.814} C_VEL
LIN {X 0,Y 447.811,Z 639.603,A -85,B 0,C 180,E1 -8743.848,E2 -8743.848} C_VEL
LIN {X 0,Y 448.422,Z 627.976,A -85,B 0,C 180,E1 -8744.639,E2 -8744.639} C_VEL
LIN {X 0,Y 448.737,Z 619.639,A -85,B 0,C 180,E1 -8745.093,E2 -8745.093} C_VEL
LIN {X 0,Y 447.775,Z 609.911,A -85,B 0,C 180,E1 -8745.56,E2 -8745.56} C_VEL
LIN {X 0,Y 446.802,Z 596.349,A -85,B 0,C 180,E1 -8746.035,E2 -8746.035} C_VEL
LIN {X 0,Y 446.11,Z 589.547,A -85,B 0,C 180,E1 -8746.225,E2 -8746.225} C_VEL
LIN {X 0,Y 446.368,Z 576.192,A -85,B 0,C 180,E1 -8749.308,E2 -8749.308} C_VEL
LIN {X 0,Y 446.66,Z 561.81,A -85,B 0,C 180,E1 -8752.675,E2 -8752.675} C_VEL
LIN {X 0,Y 447.103,Z 548.489,A -85,B 0,C 180,E1 -8755.862,E2 -8755.862} C_VEL
LIN {X 0,Y 447.523,Z 535.194,A -85,B 0,C 180,E1 -8759.133,E2 -8759.133} C_VEL
LIN {X 0,Y 448.075,Z 523.062,A -85,B 0,C 180,E1 -8762.228,E2 -8762.228} C_VEL
LIN {X 0,Y 448.729,Z 510.927,A -85,B 0,C 180,E1 -8765.469,E2 -8765.469} C_VEL
LIN {X 0,Y 448.872,Z 505.42,A -85,B 0,C 180,E1 -8767.012,E2 -8767.012} C_VEL
LIN {X 0,Y 446.992,Z 495.407,A -85,B 0,C 180,E1 -8770.139,E2 -8770.139} C_VEL
LIN {X 0,Y 446.466,Z 492.871,A -85,B 0,C 180,E1 -8771.018,E2 -8771.018} C_VEL
LIN {X 0,Y 446.404,Z 492.885,A -85,B 0,C 180,E1 -8773.846,E2 -8773.846} C_VEL
LIN {X 0,Y 446.402,Z 492.885,A -85,B 0,C 180,E1 -8776.403,E2 -8776.403} C_VEL
LIN {X 0,Y 446.43,Z 492.879,A -85,B 0,C 180,E1 -8779.083,E2 -8779.083} C_VEL
LIN {X 0,Y 446.41,Z 492.878,A -85,B 0,C 180,E1 -8782.121,E2 -8782.121} C_VEL
LIN {X 0,Y 446.425,Z 492.876,A -85,B 0,C 180,E1 -8785.477,E2 -8785.477} C_VEL
LIN {X 0,Y 446.419,Z 492.877,A -85,B 0,C 180,E1 -8788.7,E2 -8788.7} C_VEL
LIN {X 0,Y 446.488,Z 492.868,A -85,B 0,C 180,E1 -8791.822,E2 -8791.822} C_VEL
LIN {X 0,Y 446.447,Z 492.875,A -85,B 0,C 180,E1 -8794.847,E2 -8794.847} C_VEL
LIN {X 0,Y 446.452,Z 492.873,A -85,B 0,C 180,E1 -8798.245,E2 -8798.245} C_VEL
LIN {X 0,Y 446.455,Z 492.871,A -85,B 0,C 180,E1 -8801.649,E2 -8801.649} C_VEL
LIN {X 0,Y 446.511,Z 492.867,A -85,B 0,C 180,E1 -8804.48,E2 -8804.48} C_VEL
LIN {X 0,Y 446.521,Z 492.864,A -85,B 0,C 180,E1 -8808.193,E2 -8808.193} C_VEL
LIN {X 0,Y 446.604,Z 492.852,A -85,B 0,C 180,E1 -8811.858,E2 -8811.858} C_VEL
LIN {X 0,Y 446.649,Z 492.849,A -85,B 0,C 180,E1 -8814.583,E2 -8814.583} C_VEL
LIN {X 0,Y 446.667,Z 492.847,A -85,B 0,C 180,E1 -8818.197,E2 -8818.197} C_VEL
LIN {X 0,Y 446.796,Z 492.832,A -85,B 0,C 180,E1 -8820,E2 -8820} C_VEL
LIN {X 0,Y 446.695,Z 492.845,A -85,B 0,C 180,E1 -8822.706,E2 -8822.706} C_VEL
LIN {X 0,Y 446.619,Z 492.851,A -85,B 0,C 180,E1 -8826.324,E2 -8826.324} C_VEL
LIN {X 0,Y 446.541,Z 492.861,A -85,B 0,C 180,E1 -8829.056,E2 -8829.056} C_VEL
LIN {X 0,Y 446.526,Z 492.865,A -85,B 0,C 180,E1 -8832.73,E2 -8832.73} C_VEL
LIN {X 0,Y 446.5,Z 492.87,A -85,B 0,C 180,E1 -8836.228,E2 -8836.228} C_VEL
LIN {X 0,Y 446.549,Z 493.071,A -85,B 0,C 180,E1 -8838.685,E2 -8838.685} C_VEL
LIN {X 0,Y 449.97,Z 504.803,A -85,B 0,C 180,E1 -8839.503,E2 -8839.503} C_VEL
LIN {X 0,Y 449.538,Z 516.454,A -85,B 0,C 180,E1 -8840.353,E2 -8840.353} C_VEL
LIN {X 0,Y 449.03,Z 527.174,A -85,B 0,C 180,E1 -8841.34,E2 -8841.34} C_VEL
LIN {X 0,Y 448.47,Z 536.442,A -85,B 0,C 180,E1 -8842.392,E2 -8842.392} C_VEL
LIN {X 0,Y 447.973,Z 544.929,A -85,B 0,C 180,E1 -8843.582,E2 -8843.582} C_VEL
LIN {X 0,Y 447.497,Z 552.523,A -85,B 0,C 180,E1 -8844.892,E2 -8844.892} C_VEL
LIN {X 0,Y 447.11,Z 559.339,A -85,B 0,C 180,E1 -8846.366,E2 -8846.366} C_VEL
LIN {X 0,Y 446.778,Z 564.011,A -85,B 0,C 180,E1 -8847.649,E2 -8847.649} C_VEL
LIN {X 0,Y 446.525,Z 568.311,A -85,B 0,C 180,E1 -8849.204,E2 -8849.204} C_VEL
LIN {X 0,Y 446.362,Z 570.464,A -85,B 0,C 180,E1 -8850.255,E2 -8850.255} C_VEL
LIN {X 0,Y 446.213,Z 572.538,A -85,B 0,C 180,E1 -8851.731,E2 -8851.731} C_VEL
LIN {X 0,Y 446.121,Z 573.61,A -85,B 0,C 180,E1 -8853.462,E2 -8853.462} C_VEL
LIN {X 0,Y 446.097,Z 573.355,A -85,B 0,C 180,E1 -8854.992,E2 -8854.992} C_VEL
LIN {X 0,Y 446.158,Z 571.655,A -85,B 0,C 180,E1 -8856.769,E2 -8856.769} C_VEL
LIN {X 0,Y 446.323,Z 568.481,A -85,B 0,C 180,E1 -8858.5,E2 -8858.5} C_VEL
LIN {X 0,Y 446.567,Z 563.841,A -85,B 0,C 180,E1 -8860.185,E2 -8860.185} C_VEL
LIN {X 0,Y 446.847,Z 558.623,A -85,B 0,C 180,E1 -8861.602,E2 -8861.602} C_VEL
LIN {X 0,Y 447.155,Z 552.979,A -85,B 0,C 180,E1 -8862.826,E2 -8862.826} C_VEL
LIN {X 0,Y 447.568,Z 546.317,A -85,B 0,C 180,E1 -8864.015,E2 -8864.015} C_VEL
LIN {X 0,Y 448.05,Z 537.645,A -85,B 0,C 180,E1 -8865.281,E2 -8865.281} C_VEL
LIN {X 0,Y 448.539,Z 528.073,A -85,B 0,C 180,E1 -8866.415,E2 -8866.415} C_VEL
LIN {X 0,Y 449.052,Z 516.771,A -85,B 0,C 180,E1 -8867.496,E2 -8867.496} C_VEL
LIN {X 0,Y 449.546,Z 505.169,A -85,B 0,C 180,E1 -8868.361,E2 -8868.361} C_VEL
LIN {X 0,Y 448.599,Z 500.419,A -85,B 0,C 180,E1 -8868.703,E2 -8868.703} C_VEL
LIN {X 0,Y 446.432,Z 492.878,A -85,B 0,C 180,E1 -8869.236,E2 -8869.236} C_VEL
LIN {X 0,Y 446.41,Z 492.88,A -85,B 0,C 180,E1 -8872.121,E2 -8872.121} C_VEL
LIN {X 0,Y 446.434,Z 492.878,A -85,B 0,C 180,E1 -8875.477,E2 -8875.477} C_VEL
LIN {X 0,Y 446.421,Z 492.878,A -85,B 0,C 180,E1 -8878.7,E2 -8878.7} C_VEL
LIN {X 0,Y 446.49,Z 492.868,A -85,B 0,C 180,E1 -8881.821,E2 -8881.821} C_VEL
LIN {X 0,Y 446.445,Z 492.876,A -85,B 0,C 180,E1 -8884.847,E2 -8884.847} C_VEL
LIN {X 0,Y 446.454,Z 492.872,A -85,B 0,C 180,E1 -8888.245,E2 -8888.245} C_VEL
LIN {X 0,Y 446.456,Z 492.875,A -85,B 0,C 180,E1 -8891.649,E2 -8891.649} C_VEL
LIN {X 0,Y 446.513,Z 492.864,A -85,B 0,C 180,E1 -8894.48,E2 -8894.48} C_VEL
LIN {X 0,Y 446.523,Z 492.863,A -85,B 0,C 180,E1 -8898.193,E2 -8898.193} C_VEL
LIN {X 0,Y 446.518,Z 492.863,A -85,B 0,C 180,E1 -8900.373,E2 -8900.373} C_VEL
LIN {X 0,Y 445.856,Z 492.95,A -85,B 0,C 180,E1 -8901.126,E2 -8901.126} C_VEL
LIN {X 0,Y 443.017,Z 493.301,A -85,B 0,C 180,E1 -8902.35,E2 -8902.35} C_VEL
LIN {X 0,Y 440.64,Z 493.598,A -85,B 0,C 180,E1 -8903.337,E2 -8903.337} C_VEL
LIN {X 0,Y 439.657,Z 493.719,A -85,B 0,C 180,E1 -8904.1,E2 -8904.1} C_VEL
LIN {X 0,Y 439.597,Z 493.726,A -85,B 0,C 180,E1 -8904.358,E2 -8904.358} C_VEL
LIN {X 0,Y 439.638,Z 493.722,A -85,B 0,C 180,E1 -8908.168,E2 -8908.168} C_VEL
LIN {X 0,Y 439.76,Z 493.706,A -85,B 0,C 180,E1 -8910,E2 -8910} C_VEL
LIN {X 0,Y 439.637,Z 493.722,A -85,B 0,C 180,E1 -8912.749,E2 -8912.749} C_VEL
LIN {X 0,Y 439.569,Z 493.73,A -85,B 0,C 180,E1 -8916.426,E2 -8916.426} C_VEL
LIN {X 0,Y 439.501,Z 493.741,A -85,B 0,C 180,E1 -8919.202,E2 -8919.202} C_VEL
LIN {X 0,Y 439.471,Z 493.743,A -85,B 0,C 180,E1 -8922.937,E2 -8922.937} C_VEL
LIN {X 0,Y 439.451,Z 493.745,A -85,B 0,C 180,E1 -8926.348,E2 -8926.348} C_VEL
LIN {X 0,Y 439.407,Z 493.75,A -85,B 0,C 180,E1 -8929.626,E2 -8929.626} C_VEL
LIN {X 0,Y 439.368,Z 493.757,A -85,B 0,C 180,E1 -8932.575,E2 -8932.575} C_VEL
LIN {X 0,Y 439.382,Z 493.754,A -85,B 0,C 180,E1 -8935.586,E2 -8935.586} C_VEL
LIN {X 0,Y 439.404,Z 493.753,A -85,B 0,C 180,E1 -8938.674,E2 -8938.674} C_VEL
LIN {X 0,Y 439.373,Z 493.753,A -85,B 0,C 180,E1 -8942.03,E2 -8942.03} C_VEL
LIN {X 0,Y 439.395,Z 493.754,A -85,B 0,C 180,E1 -8945.339,E2 -8945.339} C_VEL
LIN {X 0,Y 439.371,Z 493.755,A -85,B 0,C 180,E1 -8948.596,E2 -8948.596} C_VEL
LIN {X 0,Y 439.371,Z 493.757,A -85,B 0,C 180,E1 -8951.253,E2 -8951.253} C_VEL
LIN {X 0,Y 439.401,Z 493.753,A -85,B 0,C 180,E1 -8954.729,E2 -8954.729} C_VEL
LIN {X 0,Y 439.387,Z 493.753,A -85,B 0,C 180,E1 -8957.794,E2 -8957.794} C_VEL
LIN {X 0,Y 439.392,Z 493.751,A -85,B 0,C 180,E1 -8960.223,E2 -8960.223} C_VEL
LIN {X 0,Y 439.375,Z 493.755,A -85,B 0,C 180,E1 -8963.712,E2 -8963.712} C_VEL
LIN {X 0,Y 439.376,Z 493.756,A -85,B 0,C 180,E1 -8967.054,E2 -8967.054} C_VEL
LIN {X 0,Y 439.386,Z 493.753,A -85,B 0,C 180,E1 -8970.274,E2 -8970.274} C_VEL
LIN {X 0,Y 439.422,Z 493.749,A -85,B 0,C 180,E1 -8973.395,E2 -8973.395} C_VEL
LIN {X 0,Y 439.386,Z 493.753,A -85,B 0,C 180,E1 -8976.429,E2 -8976.429} C_VEL
LIN {X 0,Y 439.391,Z 493.753,A -85,B 0,C 180,E1 -8979.397,E2 -8979.397} C_VEL
LIN {X 0,Y 439.428,Z 493.748,A -85,B 0,C 180,E1 -8982.309,E2 -8982.309} C_VEL
LIN {X 0,Y 439.449,Z 493.746,A -85,B 0,C 180,E1 -8985.174,E2 -8985.174} C_VEL
LIN {X 0,Y 439.486,Z 493.74,A -85,B 0,C 180,E1 -8988.001,E2 -8988.001} C_VEL
LIN {X 0,Y 439.506,Z 493.738,A -85,B 0,C 180,E1 -8991.725,E2 -8991.725} C_VEL
LIN {X 0,Y 439.611,Z 493.725,A -85,B 0,C 180,E1 -8994.495,E2 -8994.495} C_VEL
LIN {X 0,Y 439.634,Z 493.723,A -85,B 0,C 180,E1 -8998.168,E2 -8998.168} C_VEL
LIN {X 0,Y 439.761,Z 493.706,A -85,B 0,C 180,E1 -9000,E2 -9000} C_VEL
LIN {X 0,Y 439.629,Z 493.726,A -85,B 0,C 180,E1 -9002.749,E2 -9002.749} C_VEL
LIN {X 0,Y 439.568,Z 493.73,A -85,B 0,C 180,E1 -9006.426,E2 -9006.426} C_VEL
LIN {X 0,Y 439.501,Z 493.739,A -85,B 0,C 180,E1 -9009.201,E2 -9009.201} C_VEL
LIN {X 0,Y 439.506,Z 493.74,A -85,B 0,C 180,E1 -9012.726,E2 -9012.726} C_VEL
LIN {X 0,Y 439.448,Z 493.747,A -85,B 0,C 180,E1 -9016.348,E2 -9016.348} C_VEL
LIN {X 0,Y 439.404,Z 493.749,A -85,B 0,C 180,E1 -9019.626,E2 -9019.626} C_VEL
LIN {X 0,Y 439.365,Z 493.757,A -85,B 0,C 180,E1 -9022.575,E2 -9022.575} C_VEL
LIN {X 0,Y 439.381,Z 493.752,A -85,B 0,C 180,E1 -9025.586,E2 -9025.586} C_VEL
LIN {X 0,Y 439.398,Z 493.753,A -85,B 0,C 180,E1 -9028.675,E2 -9028.675} C_VEL
LIN {X 0,Y 439.37,Z 493.753,A -85,B 0,C 180,E1 -9032.03,E2 -9032.03} C_VEL
LIN {X 0,Y 439.393,Z 493.753,A -85,B 0,C 180,E1 -9035.34,E2 -9035.34} C_VEL
LIN {X 0,Y 439.371,Z 493.758,A -85,B 0,C 180,E1 -9038.596,E2 -9038.596} C_VEL
LIN {X 0,Y 439.39,Z 493.755,A -85,B 0,C 180,E1 -9041.257,E2 -9041.257} C_VEL
LIN {X 0,Y 439.4,Z 493.75,A -85,B 0,C 180,E1 -9044.729,E2 -9044.729} C_VEL
LIN {X 0,Y 439.42,Z 493.909,A -85,B 0,C 180,E1 -9047.872,E2 -9047.872} C_VEL
LIN {X 0,Y 441.332,Z 503.542,A -85,B 0,C 180,E1 -9050.886,E2 -9050.886} C_VEL
LIN {X 0,Y 442.708,Z 511.242,A -85,B 0,C 180,E1 -9053.181,E2 -9053.181} C_VEL
LIN {X 0,Y 442.144,Z 520.61,A -85,B 0,C 180,E1 -9055.747,E2 -9055.747} C_VEL
LIN {X 0,Y 441.365,Z 534.257,A -85,B 0,C 180,E1 -9059.366,E2 -9059.366} C_VEL
LIN {X 0,Y 440.59,Z 548.095,A -85,B 0,C 180,E1 -9062.929,E2 -9062.929} C_VEL
LIN {X 0,Y 440.048,Z 560.266,A -85,B 0,C 180,E1 -9065.992,E2 -9065.992} C_VEL
LIN {X 0,Y 439.557,Z 574.092,A -85,B 0,C 180,E1 -9069.405,E2 -9069.405} C_VEL
LIN {X 0,Y 439.186,Z 587.944,A -85,B 0,C 180,E1 -9072.78,E2 -9072.78} C_VEL
LIN {X 0,Y 439.081,Z 591.313,A -85,B 0,C 180,E1 -9073.595,E2 -9073.595} C_VEL
LIN {X 0,Y 440.491,Z 605.574,A -85,B 0,C 180,E1 -9074.024,E2 -9074.024} C_VEL
LIN {X 0,Y 441.43,Z 617.372,A -85,B 0,C 180,E1 -9074.533,E2 -9074.533} C_VEL
LIN {X 0,Y 441.814,Z 622.092,A -85,B 0,C 180,E1 -9074.783,E2 -9074.783} C_VEL
LIN {X 0,Y 441.247,Z 633.596,A -85,B 0,C 180,E1 -9075.472,E2 -9075.472} C_VEL
LIN {X 0,Y 440.587,Z 645.474,A -85,B 0,C 180,E1 -9076.39,E2 -9076.39} C_VEL
LIN {X 0,Y 440.121,Z 655.111,A -85,B 0,C 180,E1 -9077.317,E2 -9077.317} C_VEL
LIN {X 0,Y 439.56,Z 664.944,A -85,B 0,C 180,E1 -9078.471,E2 -9078.471} C_VEL
LIN {X 0,Y 439.167,Z 673.038,A -85,B 0,C 180,E1 -9079.628,E2 -9079.628} C_VEL
LIN {X 0,Y 438.867,Z 680.992,A -85,B 0,C 180,E1 -9081.017,E2 -9081.017} C_VEL
LIN {X 0,Y 438.759,Z 686.413,A -85,B 0,C 180,E1 -9082.175,E2 -9082.175} C_VEL
LIN {X 0,Y 438.681,Z 691.692,A -85,B 0,C 180,E1 -9083.561,E2 -9083.561} C_VEL
LIN {X 0,Y 438.732,Z 695.788,A -85,B 0,C 180,E1 -9084.946,E2 -9084.946} C_VEL
LIN {X 0,Y 438.759,Z 698.794,A -85,B 0,C 180,E1 -9086.327,E2 -9086.327} C_VEL
LIN {X 0,Y 438.742,Z 700.222,A -85,B 0,C 180,E1 -9087.246,E2 -9087.246} C_VEL
LIN {X 0,Y 438.753,Z 701.221,A -85,B 0,C 180,E1 -9088.164,E2 -9088.164} C_VEL
LIN {X 0,Y 438.919,Z 702.019,A -85,B 0,C 180,E1 -9090,E2 -9090} C_VEL
LIN {X 0,Y 438.775,Z 701.05,A -85,B 0,C 180,E1 -9091.836,E2 -9091.836} C_VEL
LIN {X 0,Y 438.77,Z 699.957,A -85,B 0,C 180,E1 -9092.754,E2 -9092.754} C_VEL
LIN {X 0,Y 438.766,Z 697.489,A -85,B 0,C 180,E1 -9094.134,E2 -9094.134} C_VEL
LIN {X 0,Y 438.729,Z 693.981,A -85,B 0,C 180,E1 -9095.516,E2 -9095.516} C_VEL
LIN {X 0,Y 438.758,Z 688.89,A -85,B 0,C 180,E1 -9097.028,E2 -9097.028} C_VEL
LIN {X 0,Y 438.873,Z 682.433,A -85,B 0,C 180,E1 -9098.519,E2 -9098.519} C_VEL
LIN {X 0,Y 439.027,Z 674.862,A -85,B 0,C 180,E1 -9099.909,E2 -9099.909} C_VEL
LIN {X 0,Y 439.482,Z 665.544,A -85,B 0,C 180,E1 -9101.297,E2 -9101.297} C_VEL
LIN {X 0,Y 440.03,Z 656.021,A -85,B 0,C 180,E1 -9102.452,E2 -9102.452} C_VEL
LIN {X 0,Y 440.342,Z 647.272,A -85,B 0,C 180,E1 -9103.334,E2 -9103.334} C_VEL
LIN {X 0,Y 441,Z 635.484,A -85,B 0,C 180,E1 -9104.301,E2 -9104.301} C_VEL
LIN {X 0,Y 441.71,Z 622.984,A -85,B 0,C 180,E1 -9105.102,E2 -9105.102} C_VEL
LIN {X 0,Y 441.507,Z 618.595,A -85,B 0,C 180,E1 -9105.346,E2 -9105.346} C_VEL
LIN {X 0,Y 440.685,Z 607.415,A -85,B 0,C 180,E1 -9105.878,E2 -9105.878} C_VEL
LIN {X 0,Y 439.588,Z 593.791,A -85,B 0,C 180,E1 -9106.354,E2 -9106.354} C_VEL
LIN {X 0,Y 439.048,Z 588.377,A -85,B 0,C 180,E1 -9106.507,E2 -9106.507} C_VEL
LIN {X 0,Y 439.318,Z 575.121,A -85,B 0,C 180,E1 -9109.63,E2 -9109.63} C_VEL
LIN {X 0,Y 439.675,Z 559.766,A -85,B 0,C 180,E1 -9113.305,E2 -9113.305} C_VEL
LIN {X 0,Y 440.139,Z 546.356,A -85,B 0,C 180,E1 -9116.595,E2 -9116.595} C_VEL
LIN {X 0,Y 440.679,Z 532.512,A -85,B 0,C 180,E1 -9120.099,E2 -9120.099} C_VEL
LIN {X 0,Y 441.175,Z 522.256,A -85,B 0,C 180,E1 -9122.795,E2 -9122.795} C_VEL
LIN {X 0,Y 441.927,Z 510.416,A -85,B 0,C 180,E1 -9126.045,E2 -9126.045} C_VEL
LIN {X 0,Y 441.796,Z 506.088,A -85,B 0,C 180,E1 -9127.308,E2 -9127.308} C_VEL
LIN {X 0,Y 439.909,Z 496.059,A -85,B 0,C 180,E1 -9130.53,E2 -9130.53} C_VEL
LIN {X 0,Y 439.427,Z 493.748,A -85,B 0,C 180,E1 -9131.342,E2 -9131.342} C_VEL
LIN {X 0,Y 439.404,Z 493.756,A -85,B 0,C 180,E1 -9135.271,E2 -9135.271} C_VEL
LIN {X 0,Y 439.391,Z 493.757,A -85,B 0,C 180,E1 -9138.743,E2 -9138.743} C_VEL
LIN {X 0,Y 439.376,Z 493.754,A -85,B 0,C 180,E1 -9141.608,E2 -9141.608} C_VEL
LIN {X 0,Y 439.398,Z 493.755,A -85,B 0,C 180,E1 -9144.844,E2 -9144.844} C_VEL
LIN {X 0,Y 439.375,Z 493.753,A -85,B 0,C 180,E1 -9148.14,E2 -9148.14} C_VEL
LIN {X 0,Y 439.436,Z 493.747,A -85,B 0,C 180,E1 -9151.598,E2 -9151.598} C_VEL
LIN {X 0,Y 439.401,Z 493.751,A -85,B 0,C 180,E1 -9154.415,E2 -9154.415} C_VEL
LIN {X 0,Y 439.367,Z 493.757,A -85,B 0,C 180,E1 -9157.425,E2 -9157.425} C_VEL
LIN {X 0,Y 439.444,Z 493.747,A -85,B 0,C 180,E1 -9160.663,E2 -9160.663} C_VEL
LIN {X 0,Y 439.466,Z 493.744,A -85,B 0,C 180,E1 -9164.225,E2 -9164.225} C_VEL
LIN {X 0,Y 439.487,Z 493.74,A -85,B 0,C 180,E1 -9168.002,E2 -9168.002} C_VEL
LIN {X 0,Y 439.552,Z 493.73,A -85,B 0,C 180,E1 -9171.727,E2 -9171.727} C_VEL
LIN {X 0,Y 439.624,Z 493.725,A -85,B 0,C 180,E1 -9174.496,E2 -9174.496} C_VEL
LIN {X 0,Y 439.637,Z 493.722,A -85,B 0,C 180,E1 -9178.168,E2 -9178.168} C_VEL
LIN {X 0,Y 439.765,Z 493.707,A -85,B 0,C 180,E1 -9180,E2 -9180} C_VEL
LIN {X 0,Y 439.644,Z 493.723,A -85,B 0,C 180,E1 -9182.749,E2 -9182.749} C_VEL
LIN {X 0,Y 439.57,Z 493.729,A -85,B 0,C 180,E1 -9186.426,E2 -9186.426} C_VEL
LIN {X 0,Y 439.503,Z 493.738,A -85,B 0,C 180,E1 -9189.202,E2 -9189.202} C_VEL
LIN {X 0,Y 439.47,Z 493.744,A -85,B 0,C 180,E1 -9192.938,E2 -9192.938} C_VEL
LIN {X 0,Y 439.469,Z 493.746,A -85,B 0,C 180,E1 -9196.356,E2 -9196.356} C_VEL
LIN {X 0,Y 439.445,Z 493.753,A -85,B 0,C 180,E1 -9198.383,E2 -9198.383} C_VEL
LIN {X 0,Y 442.768,Z 504.915,A -85,B 0,C 180,E1 -9199.178,E2 -9199.178} C_VEL
LIN {X 0,Y 443.224,Z 506.496,A -85,B 0,C 180,E1 -9199.304,E2 -9199.304} C_VEL
LIN {X 0,Y 442.709,Z 518.485,A -85,B 0,C 180,E1 -9200.204,E2 -9200.204} C_VEL
LIN {X 0,Y 442.22,Z 528.69,A -85,B 0,C 180,E1 -9201.172,E2 -9201.172} C_VEL
LIN {X 0,Y 441.619,Z 537.617,A -85,B 0,C 180,E1 -9202.208,E2 -9202.208} C_VEL
LIN {X 0,Y 441.073,Z 546.434,A -85,B 0,C 180,E1 -9203.475,E2 -9203.475} C_VEL
LIN {X 0,Y 440.586,Z 553.549,A -85,B 0,C 180,E1 -9204.729,E2 -9204.729} C_VEL
LIN {X 0,Y 440.149,Z 560.663,A -85,B 0,C 180,E1 -9206.302,E2 -9206.302} C_VEL
LIN {X 0,Y 439.816,Z 565.286,A -85,B 0,C 180,E1 -9207.607,E2 -9207.607} C_VEL
LIN {X 0,Y 439.545,Z 569.513,A -85,B 0,C 180,E1 -9209.188,E2 -9209.188} C_VEL
LIN {X 0,Y 439.294,Z 572.475,A -85,B 0,C 180,E1 -9210.794,E2 -9210.794} C_VEL
LIN {X 0,Y 439.169,Z 573.869,A -85,B 0,C 180,E1 -9211.988,E2 -9211.988} C_VEL
LIN {X 0,Y 439.097,Z 574.662,A -85,B 0,C 180,E1 -9213.665,E2 -9213.665} C_VEL
LIN {X 0,Y 439.094,Z 574.203,A -85,B 0,C 180,E1 -9215.284,E2 -9215.284} C_VEL
LIN {X 0,Y 439.138,Z 572.604,A -85,B 0,C 180,E1 -9216.85,E2 -9216.85} C_VEL
LIN {X 0,Y 439.324,Z 569.382,A -85,B 0,C 180,E1 -9218.602,E2 -9218.602} C_VEL
LIN {X 0,Y 439.607,Z 564.541,A -85,B 0,C 180,E1 -9220.36,E2 -9220.36} C_VEL
LIN {X 0,Y 439.864,Z 559.698,A -85,B 0,C 180,E1 -9221.684,E2 -9221.684} C_VEL
LIN {X 0,Y 440.282,Z 552.958,A -85,B 0,C 180,E1 -9223.145,E2 -9223.145} C_VEL
LIN {X 0,Y 440.788,Z 544.791,A -85,B 0,C 180,E1 -9224.552,E2 -9224.552} C_VEL
LIN {X 0,Y 441.295,Z 536.002,A -85,B 0,C 180,E1 -9225.78,E2 -9225.78} C_VEL
LIN {X 0,Y 441.783,Z 526.755,A -85,B 0,C 180,E1 -9226.838,E2 -9226.838} C_VEL
LIN {X 0,Y 442.277,Z 516.284,A -85,B 0,C 180,E1 -9227.808,E2 -9227.808} C_VEL
LIN {X 0,Y 442.676,Z 505.77,A -85,B 0,C 180,E1 -9228.595,E2 -9228.595} C_VEL
LIN {X 0,Y 439.397,Z 493.754,A -85,B 0,C 180,E1 -9229.475,E2 -9229.475} C_VEL
LIN {X 0,Y 439.35,Z 493.761,A -85,B 0,C 180,E1 -9232.565,E2 -9232.565} C_VEL
LIN {X 0,Y 439.403,Z 493.75,A -85,B 0,C 180,E1 -9234.844,E2 -9234.844} C_VEL
LIN {X 0,Y 439.378,Z 493.755,A -85,B 0,C 180,E1 -9238.14,E2 -9238.14} C_VEL
LIN {X 0,Y 439.438,Z 493.748,A -85,B 0,C 180,E1 -9241.598,E2 -9241.598} C_VEL
LIN {X 0,Y 439.392,Z 493.752,A -85,B 0,C 180,E1 -9244.414,E2 -9244.414} C_VEL
LIN {X 0,Y 439.369,Z 493.759,A -85,B 0,C 180,E1 -9247.425,E2 -9247.425} C_VEL
LIN {X 0,Y 439.446,Z 493.746,A -85,B 0,C 180,E1 -9250.663,E2 -9250.663} C_VEL
LIN {X 0,Y 439.467,Z 493.742,A -85,B 0,C 180,E1 -9254.224,E2 -9254.224} C_VEL
LIN {X 0,Y 439.489,Z 493.74,A -85,B 0,C 180,E1 -9258.001,E2 -9258.001} C_VEL
LIN {X 0,Y 439.509,Z 493.739,A -85,B 0,C 180,E1 -9261.725,E2 -9261.725} C_VEL
LIN {X 0,Y 439.597,Z 493.726,A -85,B 0,C 180,E1 -9264.358,E2 -9264.358} C_VEL
LIN {X 0,Y 438.995,Z 493.804,A -85,B 0,C 180,E1 -9265.122,E2 -9265.122} C_VEL
LIN {X 0,Y 436.194,Z 494.153,A -85,B 0,C 180,E1 -9266.364,E2 -9266.364} C_VEL
LIN {X 0,Y 433.764,Z 494.455,A -85,B 0,C 180,E1 -9267.366,E2 -9267.366} C_VEL
LIN {X 0,Y 432.682,Z 494.588,A -85,B 0,C 180,E1 -9268.14,E2 -9268.14} C_VEL
LIN {X 0,Y 432.576,Z 494.6,A -85,B 0,C 180,E1 -9268.402,E2 -9268.402} C_VEL
LIN {X 0,Y 432.729,Z 494.582,A -85,B 0,C 180,E1 -9270,E2 -9270} C_VEL
LIN {X 0,Y 432.589,Z 494.6,A -85,B 0,C 180,E1 -9272.794,E2 -9272.794} C_VEL
LIN {X 0,Y 432.583,Z 494.603,A -85,B 0,C 180,E1 -9275.594,E2 -9275.594} C_VEL
LIN {X 0,Y 432.469,Z 494.613,A -85,B 0,C 180,E1 -9278.41,E2 -9278.41} C_VEL
LIN {X 0,Y 432.464,Z 494.614,A -85,B 0,C 180,E1 -9282.196,E2 -9282.196} C_VEL
LIN {X 0,Y 432.435,Z 494.619,A -85,B 0,C 180,E1 -9286.039,E2 -9286.039} C_VEL
LIN {X 0,Y 432.391,Z 494.625,A -85,B 0,C 180,E1 -9289.485,E2 -9289.485} C_VEL
LIN {X 0,Y 432.322,Z 494.634,A -85,B 0,C 180,E1 -9292.964,E2 -9292.964} C_VEL
LIN {X 0,Y 432.342,Z 494.632,A -85,B 0,C 180,E1 -9295.002,E2 -9295.002} C_VEL
LIN {X 0,Y 432.352,Z 494.629,A -85,B 0,C 180,E1 -9298.125,E2 -9298.125} C_VEL
LIN {X 0,Y 432.324,Z 494.635,A -85,B 0,C 180,E1 -9301.346,E2 -9301.346} C_VEL
LIN {X 0,Y 432.341,Z 494.633,A -85,B 0,C 180,E1 -9304.677,E2 -9304.677} C_VEL
LIN {X 0,Y 432.335,Z 494.63,A -85,B 0,C 180,E1 -9308.15,E2 -9308.15} C_VEL
LIN {X 0,Y 432.315,Z 494.635,A -85,B 0,C 180,E1 -9311.598,E2 -9311.598} C_VEL
LIN {X 0,Y 432.337,Z 494.63,A -85,B 0,C 180,E1 -9314.347,E2 -9314.347} C_VEL
LIN {X 0,Y 432.319,Z 494.634,A -85,B 0,C 180,E1 -9317.016,E2 -9317.016} C_VEL
LIN {X 0,Y 432.335,Z 494.63,A -85,B 0,C 180,E1 -9319.821,E2 -9319.821} C_VEL
LIN {X 0,Y 432.307,Z 494.636,A -85,B 0,C 180,E1 -9323.021,E2 -9323.021} C_VEL
LIN {X 0,Y 432.362,Z 494.626,A -85,B 0,C 180,E1 -9325.996,E2 -9325.996} C_VEL
LIN {X 0,Y 432.351,Z 494.631,A -85,B 0,C 180,E1 -9329.489,E2 -9329.489} C_VEL
LIN {X 0,Y 432.388,Z 494.627,A -85,B 0,C 180,E1 -9332.928,E2 -9332.928} C_VEL
LIN {X 0,Y 432.369,Z 494.626,A -85,B 0,C 180,E1 -9336.023,E2 -9336.023} C_VEL
LIN {X 0,Y 432.353,Z 494.631,A -85,B 0,C 180,E1 -9339.046,E2 -9339.046} C_VEL
LIN {X 0,Y 432.376,Z 494.626,A -85,B 0,C 180,E1 -9342.011,E2 -9342.011} C_VEL
LIN {X 0,Y 432.397,Z 494.626,A -85,B 0,C 180,E1 -9344.926,E2 -9344.926} C_VEL
LIN {X 0,Y 432.462,Z 494.615,A -85,B 0,C 180,E1 -9347.803,E2 -9347.803} C_VEL
LIN {X 0,Y 432.466,Z 494.616,A -85,B 0,C 180,E1 -9351.59,E2 -9351.59} C_VEL
LIN {X 0,Y 432.587,Z 494.6,A -85,B 0,C 180,E1 -9354.406,E2 -9354.406} C_VEL
LIN {X 0,Y 432.603,Z 494.598,A -85,B 0,C 180,E1 -9358.138,E2 -9358.138} C_VEL
LIN {X 0,Y 432.73,Z 494.582,A -85,B 0,C 180,E1 -9360,E2 -9360} C_VEL
LIN {X 0,Y 432.58,Z 494.604,A -85,B 0,C 180,E1 -9362.793,E2 -9362.793} C_VEL
LIN {X 0,Y 432.581,Z 494.601,A -85,B 0,C 180,E1 -9365.594,E2 -9365.594} C_VEL
LIN {X 0,Y 432.485,Z 494.613,A -85,B 0,C 180,E1 -9368.41,E2 -9368.41} C_VEL
LIN {X 0,Y 432.483,Z 494.613,A -85,B 0,C 180,E1 -9372.196,E2 -9372.196} C_VEL
LIN {X 0,Y 432.432,Z 494.619,A -85,B 0,C 180,E1 -9376.039,E2 -9376.039} C_VEL
LIN {X 0,Y 432.388,Z 494.623,A -85,B 0,C 180,E1 -9379.485,E2 -9379.485} C_VEL
LIN {X 0,Y 432.319,Z 494.635,A -85,B 0,C 180,E1 -9382.964,E2 -9382.964} C_VEL
LIN {X 0,Y 432.34,Z 494.633,A -85,B 0,C 180,E1 -9385.002,E2 -9385.002} C_VEL
LIN {X 0,Y 432.345,Z 494.631,A -85,B 0,C 180,E1 -9388.126,E2 -9388.126} C_VEL
LIN {X 0,Y 432.322,Z 494.632,A -85,B 0,C 180,E1 -9391.346,E2 -9391.346} C_VEL
LIN {X 0,Y 432.339,Z 494.632,A -85,B 0,C 180,E1 -9394.677,E2 -9394.677} C_VEL
LIN {X 0,Y 432.334,Z 494.63,A -85,B 0,C 180,E1 -9398.15,E2 -9398.15} C_VEL
LIN {X 0,Y 432.334,Z 494.634,A -85,B 0,C 180,E1 -9401.602,E2 -9401.602} C_VEL
LIN {X 0,Y 432.334,Z 494.631,A -85,B 0,C 180,E1 -9404.347,E2 -9404.347} C_VEL
LIN {X 0,Y 432.362,Z 494.806,A -85,B 0,C 180,E1 -9407.564,E2 -9407.564} C_VEL
LIN {X 0,Y 434.248,Z 504.227,A -85,B 0,C 180,E1 -9410.569,E2 -9410.569} C_VEL
LIN {X 0,Y 435.684,Z 511.629,A -85,B 0,C 180,E1 -9412.834,E2 -9412.834} C_VEL
LIN {X 0,Y 435.512,Z 517.465,A -85,B 0,C 180,E1 -9414.483,E2 -9414.483} C_VEL
LIN {X 0,Y 434.657,Z 529.431,A -85,B 0,C 180,E1 -9417.752,E2 -9417.752} C_VEL
LIN {X 0,Y 434.062,Z 539.404,A -85,B 0,C 180,E1 -9420.407,E2 -9420.407} C_VEL
LIN {X 0,Y 433.297,Z 553.336,A -85,B 0,C 180,E1 -9424.028,E2 -9424.028} C_VEL
LIN {X 0,Y 432.801,Z 565.242,A -85,B 0,C 180,E1 -9427.063,E2 -9427.063} C_VEL
LIN {X 0,Y 432.289,Z 579.135,A -85,B 0,C 180,E1 -9430.552,E2 -9430.552} C_VEL
LIN {X 0,Y 432.047,Z 590.349,A -85,B 0,C 180,E1 -9433.324,E2 -9433.324} C_VEL
LIN {X 0,Y 433.574,Z 606.147,A -85,B 0,C 180,E1 -9433.832,E2 -9433.832} C_VEL
LIN {X 0,Y 434.491,Z 618.469,A -85,B 0,C 180,E1 -9434.4,E2 -9434.4} C_VEL
LIN {X 0,Y 434.806,Z 623.001,A -85,B 0,C 180,E1 -9434.652,E2 -9434.652} C_VEL
LIN {X 0,Y 434.148,Z 635.615,A -85,B 0,C 180,E1 -9435.468,E2 -9435.468} C_VEL
LIN {X 0,Y 433.458,Z 647.432,A -85,B 0,C 180,E1 -9436.45,E2 -9436.45} C_VEL
LIN {X 0,Y 433.052,Z 655.04,A -85,B 0,C 180,E1 -9437.225,E2 -9437.225} C_VEL
LIN {X 0,Y 432.458,Z 665.605,A -85,B 0,C 180,E1 -9438.517,E2 -9438.517} C_VEL
LIN {X 0,Y 431.971,Z 674.786,A -85,B 0,C 180,E1 -9439.927,E2 -9439.927} C_VEL
LIN {X 0,Y 431.773,Z 682.219,A -85,B 0,C 180,E1 -9441.341,E2 -9441.341} C_VEL
LIN {X 0,Y 431.635,Z 687.244,A -85,B 0,C 180,E1 -9442.516,E2 -9442.516} C_VEL
LIN {X 0,Y 431.647,Z 692.133,A -85,B 0,C 180,E1 -9443.925,E2 -9443.925} C_VEL
LIN {X 0,Y 431.692,Z 695.862,A -85,B 0,C 180,E1 -9445.331,E2 -9445.331} C_VEL
LIN {X 0,Y 431.721,Z 697.776,A -85,B 0,C 180,E1 -9446.267,E2 -9446.267} C_VEL
LIN {X 0,Y 431.701,Z 699.206,A -85,B 0,C 180,E1 -9447.201,E2 -9447.201} C_VEL
LIN {X 0,Y 431.718,Z 700.204,A -85,B 0,C 180,E1 -9448.134,E2 -9448.134} C_VEL
LIN {X 0,Y 431.901,Z 701.002,A -85,B 0,C 180,E1 -9450,E2 -9450} C_VEL
LIN {X 0,Y 431.741,Z 700.024,A -85,B 0,C 180,E1 -9451.866,E2 -9451.866} C_VEL
LIN {X 0,Y 431.729,Z 698.927,A -85,B 0,C 180,E1 -9452.799,E2 -9452.799} C_VEL
LIN {X 0,Y 431.735,Z 696.456,A -85,B 0,C 180,E1 -9454.201,E2 -9454.201} C_VEL
LIN {X 0,Y 431.667,Z 692.94,A -85,B 0,C 180,E1 -9455.606,E2 -9455.606} C_VEL
LIN {X 0,Y 431.689,Z 688.492,A -85,B 0,C 180,E1 -9456.967,E2 -9456.967} C_VEL
LIN {X 0,Y 431.791,Z 682.467,A -85,B 0,C 180,E1 -9458.424,E2 -9458.424} C_VEL
LIN {X 0,Y 431.95,Z 675.196,A -85,B 0,C 180,E1 -9459.837,E2 -9459.837} C_VEL
LIN {X 0,Y 432.363,Z 666.17,A -85,B 0,C 180,E1 -9461.248,E2 -9461.248} C_VEL
LIN {X 0,Y 432.917,Z 657.043,A -85,B 0,C 180,E1 -9462.415,E2 -9462.415} C_VEL
LIN {X 0,Y 433.257,Z 648.38,A -85,B 0,C 180,E1 -9463.341,E2 -9463.341} C_VEL
LIN {X 0,Y 433.904,Z 637.495,A -85,B 0,C 180,E1 -9464.301,E2 -9464.301} C_VEL
LIN {X 0,Y 434.622,Z 625.953,A -85,B 0,C 180,E1 -9465.115,E2 -9465.115} C_VEL
LIN {X 0,Y 434.717,Z 620.995,A -85,B 0,C 180,E1 -9465.411,E2 -9465.411} C_VEL
LIN {X 0,Y 433.905,Z 610.246,A -85,B 0,C 180,E1 -9465.983,E2 -9465.983} C_VEL
LIN {X 0,Y 432.998,Z 596.948,A -85,B 0,C 180,E1 -9466.51,E2 -9466.51} C_VEL
LIN {X 0,Y 431.987,Z 587.166,A -85,B 0,C 180,E1 -9466.812,E2 -9466.812} C_VEL
LIN {X 0,Y 432.259,Z 573.037,A -85,B 0,C 180,E1 -9470.212,E2 -9470.212} C_VEL
LIN {X 0,Y 432.611,Z 559.787,A -85,B 0,C 180,E1 -9473.454,E2 -9473.454} C_VEL
LIN {X 0,Y 433.068,Z 548.01,A -85,B 0,C 180,E1 -9476.399,E2 -9476.399} C_VEL
LIN {X 0,Y 433.588,Z 534.447,A -85,B 0,C 180,E1 -9479.896,E2 -9479.896} C_VEL
LIN {X 0,Y 434.213,Z 522.934,A -85,B 0,C 180,E1 -9482.977,E2 -9482.977} C_VEL
LIN {X 0,Y 435.029,Z 510.921,A -85,B 0,C 180,E1 -9486.354,E2 -9486.354} C_VEL
LIN {X 0,Y 434.727,Z 506.767,A -85,B 0,C 180,E1 -9487.612,E2 -9487.612} C_VEL
LIN {X 0,Y 433.083,Z 498.053,A -85,B 0,C 180,E1 -9490.475,E2 -9490.475} C_VEL
LIN {X 0,Y 432.387,Z 494.627,A -85,B 0,C 180,E1 -9491.693,E2 -9491.693} C_VEL
LIN {X 0,Y 432.336,Z 494.636,A -85,B 0,C 180,E1 -9494.348,E2 -9494.348} C_VEL
LIN {X 0,Y 432.323,Z 494.637,A -85,B 0,C 180,E1 -9497.016,E2 -9497.016} C_VEL
LIN {X 0,Y 432.336,Z 494.634,A -85,B 0,C 180,E1 -9499.821,E2 -9499.821} C_VEL
LIN {X 0,Y 432.307,Z 494.636,A -85,B 0,C 180,E1 -9503.022,E2 -9503.022} C_VEL
LIN {X 0,Y 432.36,Z 494.628,A -85,B 0,C 180,E1 -9505.997,E2 -9505.997} C_VEL
LIN {X 0,Y 432.351,Z 494.63,A -85,B 0,C 180,E1 -9509.49,E2 -9509.49} C_VEL
LIN {X 0,Y 432.394,Z 494.622,A -85,B 0,C 180,E1 -9512.928,E2 -9512.928} C_VEL
LIN {X 0,Y 432.371,Z 494.624,A -85,B 0,C 180,E1 -9516.023,E2 -9516.023} C_VEL
LIN {X 0,Y 432.354,Z 494.626,A -85,B 0,C 180,E1 -9519.046,E2 -9519.046} C_VEL
LIN {X 0,Y 432.377,Z 494.624,A -85,B 0,C 180,E1 -9522.011,E2 -9522.011} C_VEL
LIN {X 0,Y 432.399,Z 494.621,A -85,B 0,C 180,E1 -9524.927,E2 -9524.927} C_VEL
LIN {X 0,Y 432.463,Z 494.615,A -85,B 0,C 180,E1 -9527.804,E2 -9527.804} C_VEL
LIN {X 0,Y 432.496,Z 494.609,A -85,B 0,C 180,E1 -9531.591,E2 -9531.591} C_VEL
LIN {X 0,Y 432.601,Z 494.599,A -85,B 0,C 180,E1 -9534.406,E2 -9534.406} C_VEL
LIN {X 0,Y 432.606,Z 494.598,A -85,B 0,C 180,E1 -9538.138,E2 -9538.138} C_VEL
LIN {X 0,Y 432.735,Z 494.583,A -85,B 0,C 180,E1 -9540,E2 -9540} C_VEL
LIN {X 0,Y 432.596,Z 494.601,A -85,B 0,C 180,E1 -9542.794,E2 -9542.794} C_VEL
LIN {X 0,Y 432.584,Z 494.601,A -85,B 0,C 180,E1 -9545.594,E2 -9545.594} C_VEL
LIN {X 0,Y 432.487,Z 494.612,A -85,B 0,C 180,E1 -9548.41,E2 -9548.41} C_VEL
LIN {X 0,Y 432.464,Z 494.619,A -85,B 0,C 180,E1 -9552.197,E2 -9552.197} C_VEL
LIN {X 0,Y 432.443,Z 494.621,A -85,B 0,C 180,E1 -9556.039,E2 -9556.039} C_VEL
LIN {X 0,Y 432.409,Z 494.63,A -85,B 0,C 180,E1 -9558.08,E2 -9558.08} C_VEL
LIN {X 0,Y 436.266,Z 507.506,A -85,B 0,C 180,E1 -9559.04,E2 -9559.04} C_VEL
LIN {X 0,Y 436.122,Z 515.836,A -85,B 0,C 180,E1 -9559.658,E2 -9559.658} C_VEL
LIN {X 0,Y 435.57,Z 526.708,A -85,B 0,C 180,E1 -9560.634,E2 -9560.634} C_VEL
LIN {X 0,Y 434.908,Z 537.219,A -85,B 0,C 180,E1 -9561.819,E2 -9561.819} C_VEL
LIN {X 0,Y 434.302,Z 546.374,A -85,B 0,C 180,E1 -9563.106,E2 -9563.106} C_VEL
LIN {X 0,Y 433.779,Z 553.547,A -85,B 0,C 180,E1 -9564.352,E2 -9564.352} C_VEL
LIN {X 0,Y 433.359,Z 559.888,A -85,B 0,C 180,E1 -9565.711,E2 -9565.711} C_VEL
LIN {X 0,Y 432.963,Z 564.865,A -85,B 0,C 180,E1 -9567.034,E2 -9567.034} C_VEL
LIN {X 0,Y 432.631,Z 569.628,A -85,B 0,C 180,E1 -9568.691,E2 -9568.691} C_VEL
LIN {X 0,Y 432.348,Z 572.827,A -85,B 0,C 180,E1 -9570.26,E2 -9570.26} C_VEL
LIN {X 0,Y 432.228,Z 574.315,A -85,B 0,C 180,E1 -9571.354,E2 -9571.354} C_VEL
LIN {X 0,Y 432.115,Z 575.298,A -85,B 0,C 180,E1 -9572.461,E2 -9572.461} C_VEL
LIN {X 0,Y 432.068,Z 575.715,A -85,B 0,C 180,E1 -9573.945,E2 -9573.945} C_VEL
LIN {X 0,Y 432.075,Z 575.034,A -85,B 0,C 180,E1 -9575.581,E2 -9575.581} C_VEL
LIN {X 0,Y 432.144,Z 573.201,A -85,B 0,C 180,E1 -9577.165,E2 -9577.165} C_VEL
LIN {X 0,Y 432.317,Z 570.272,A -85,B 0,C 180,E1 -9578.71,E2 -9578.71} C_VEL
LIN {X 0,Y 432.573,Z 566.246,A -85,B 0,C 180,E1 -9580.216,E2 -9580.216} C_VEL
LIN {X 0,Y 432.87,Z 560.906,A -85,B 0,C 180,E1 -9581.734,E2 -9581.734} C_VEL
LIN {X 0,Y 433.353,Z 553.752,A -85,B 0,C 180,E1 -9583.31,E2 -9583.31} C_VEL
LIN {X 0,Y 433.845,Z 545.892,A -85,B 0,C 180,E1 -9584.683,E2 -9584.683} C_VEL
LIN {X 0,Y 434.412,Z 536.501,A -85,B 0,C 180,E1 -9586.013,E2 -9586.013} C_VEL
LIN {X 0,Y 434.979,Z 526.31,A -85,B 0,C 180,E1 -9587.168,E2 -9587.168} C_VEL
LIN {X 0,Y 435.521,Z 515.258,A -85,B 0,C 180,E1 -9588.175,E2 -9588.175} C_VEL
LIN {X 0,Y 435.835,Z 507.359,A -85,B 0,C 180,E1 -9588.766,E2 -9588.766} C_VEL
LIN {X 0,Y 432.679,Z 496.057,A -85,B 0,C 180,E1 -9589.594,E2 -9589.594} C_VEL
LIN {X 0,Y 432.35,Z 494.632,A -85,B 0,C 180,E1 -9589.7,E2 -9589.7} C_VEL
LIN {X 0,Y 432.309,Z 494.636,A -85,B 0,C 180,E1 -9593.022,E2 -9593.022} C_VEL
LIN {X 0,Y 432.364,Z 494.627,A -85,B 0,C 180,E1 -9595.997,E2 -9595.997} C_VEL
LIN {X 0,Y 432.352,Z 494.631,A -85,B 0,C 180,E1 -9599.49,E2 -9599.49} C_VEL
LIN {X 0,Y 432.391,Z 494.625,A -85,B 0,C 180,E1 -9602.928,E2 -9602.928} C_VEL
LIN {X 0,Y 432.372,Z 494.627,A -85,B 0,C 180,E1 -9606.023,E2 -9606.023} C_VEL
LIN {X 0,Y 432.356,Z 494.631,A -85,B 0,C 180,E1 -9609.046,E2 -9609.046} C_VEL
LIN {X 0,Y 432.365,Z 494.628,A -85,B 0,C 180,E1 -9612.01,E2 -9612.01} C_VEL
LIN {X 0,Y 432.399,Z 494.625,A -85,B 0,C 180,E1 -9614.926,E2 -9614.926} C_VEL
LIN {X 0,Y 432.465,Z 494.616,A -85,B 0,C 180,E1 -9617.803,E2 -9617.803} C_VEL
LIN {X 0,Y 432.469,Z 494.616,A -85,B 0,C 180,E1 -9621.59,E2 -9621.59} C_VEL
LIN {X 0,Y 432.584,Z 494.599,A -85,B 0,C 180,E1 -9624.406,E2 -9624.406} C_VEL
LIN {X 0,Y 432.608,Z 494.597,A -85,B 0,C 180,E1 -9628.138,E2 -9628.138} C_VEL
LIN {X 0,Y 432.576,Z 494.6,A -85,B 0,C 180,E1 -9628.402,E2 -9628.402} C_VEL
LIN {X 0,Y 431.865,Z 494.692,A -85,B 0,C 180,E1 -9629.179,E2 -9629.179} C_VEL
LIN {X 0,Y 429.02,Z 495.043,A -85,B 0,C 180,E1 -9630.443,E2 -9630.443} C_VEL
LIN {X 0,Y 426.643,Z 495.342,A -85,B 0,C 180,E1 -9631.462,E2 -9631.462} C_VEL
LIN {X 0,Y 425.625,Z 495.466,A -85,B 0,C 180,E1 -9632.25,E2 -9632.25} C_VEL
LIN {X 0,Y 425.541,Z 495.476,A -85,B 0,C 180,E1 -9632.516,E2 -9632.516} C_VEL
LIN {X 0,Y 425.537,Z 495.48,A -85,B 0,C 180,E1 -9635.687,E2 -9635.687} C_VEL
LIN {X 0,Y 425.413,Z 495.493,A -85,B 0,C 180,E1 -9638.551,E2 -9638.551} C_VEL
LIN {X 0,Y 425.417,Z 495.492,A -85,B 0,C 180,E1 -9642.402,E2 -9642.402} C_VEL
LIN {X 0,Y 425.393,Z 495.496,A -85,B 0,C 180,E1 -9646.312,E2 -9646.312} C_VEL
LIN {X 0,Y 425.333,Z 495.503,A -85,B 0,C 180,E1 -9649.635,E2 -9649.635} C_VEL
LIN {X 0,Y 425.308,Z 495.509,A -85,B 0,C 180,E1 -9653.365,E2 -9653.365} C_VEL
LIN {X 0,Y 425.305,Z 495.506,A -85,B 0,C 180,E1 -9656.498,E2 -9656.498} C_VEL
LIN {X 0,Y 425.29,Z 495.51,A -85,B 0,C 180,E1 -9659.72,E2 -9659.72} C_VEL
LIN {X 0,Y 425.286,Z 495.512,A -85,B 0,C 180,E1 -9663.048,E2 -9663.048} C_VEL
LIN {X 0,Y 425.284,Z 495.509,A -85,B 0,C 180,E1 -9665.928,E2 -9665.928} C_VEL
LIN {X 0,Y 425.268,Z 495.514,A -85,B 0,C 180,E1 -9669.038,E2 -9669.038} C_VEL
LIN {X 0,Y 425.264,Z 495.512,A -85,B 0,C 180,E1 -9672.655,E2 -9672.655} C_VEL
LIN {X 0,Y 425.288,Z 495.51,A -85,B 0,C 180,E1 -9675.283,E2 -9675.283} C_VEL
LIN {X 0,Y 425.27,Z 495.511,A -85,B 0,C 180,E1 -9678.62,E2 -9678.62} C_VEL
LIN {X 0,Y 425.295,Z 495.51,A -85,B 0,C 180,E1 -9681.1,E2 -9681.1} C_VEL
LIN {X 0,Y 425.302,Z 495.508,A -85,B 0,C 180,E1 -9684.664,E2 -9684.664} C_VEL
LIN {X 0,Y 425.268,Z 495.511,A -85,B 0,C 180,E1 -9688.073,E2 -9688.073} C_VEL
LIN {X 0,Y 425.334,Z 495.504,A -85,B 0,C 180,E1 -9691.368,E2 -9691.368} C_VEL
LIN {X 0,Y 425.287,Z 495.511,A -85,B 0,C 180,E1 -9694.554,E2 -9694.554} C_VEL
LIN {X 0,Y 425.287,Z 495.51,A -85,B 0,C 180,E1 -9696.633,E2 -9696.633} C_VEL
LIN {X 0,Y 425.298,Z 495.508,A -85,B 0,C 180,E1 -9699.694,E2 -9699.694} C_VEL
LIN {X 0,Y 425.342,Z 495.503,A -85,B 0,C 180,E1 -9702.697,E2 -9702.697} C_VEL
LIN {X 0,Y 425.35,Z 495.502,A -85,B 0,C 180,E1 -9705.65,E2 -9705.65} C_VEL
LIN {X 0,Y 425.353,Z 495.501,A -85,B 0,C 180,E1 -9708.564,E2 -9708.564} C_VEL
LIN {X 0,Y 425.41,Z 495.495,A -85,B 0,C 180,E1 -9711.449,E2 -9711.449} C_VEL
LIN {X 0,Y 425.542,Z 495.478,A -85,B 0,C 180,E1 -9714.313,E2 -9714.313} C_VEL
LIN {X 0,Y 425.573,Z 495.474,A -85,B 0,C 180,E1 -9718.107,E2 -9718.107} C_VEL
LIN {X 0,Y 425.7,Z 495.457,A -85,B 0,C 180,E1 -9720,E2 -9720} C_VEL
LIN {X 0,Y 425.534,Z 495.481,A -85,B 0,C 180,E1 -9722.84,E2 -9722.84} C_VEL
LIN {X 0,Y 425.535,Z 495.478,A -85,B 0,C 180,E1 -9725.687,E2 -9725.687} C_VEL
LIN {X 0,Y 425.439,Z 495.492,A -85,B 0,C 180,E1 -9728.55,E2 -9728.55} C_VEL
LIN {X 0,Y 425.432,Z 495.491,A -85,B 0,C 180,E1 -9732.401,E2 -9732.401} C_VEL
LIN {X 0,Y 425.39,Z 495.498,A -85,B 0,C 180,E1 -9736.312,E2 -9736.312} C_VEL
LIN {X 0,Y 425.33,Z 495.502,A -85,B 0,C 180,E1 -9739.635,E2 -9739.635} C_VEL
LIN {X 0,Y 425.306,Z 495.508,A -85,B 0,C 180,E1 -9743.365,E2 -9743.365} C_VEL
LIN {X 0,Y 425.303,Z 495.509,A -85,B 0,C 180,E1 -9746.498,E2 -9746.498} C_VEL
LIN {X 0,Y 425.287,Z 495.509,A -85,B 0,C 180,E1 -9749.72,E2 -9749.72} C_VEL
LIN {X 0,Y 425.283,Z 495.511,A -85,B 0,C 180,E1 -9753.048,E2 -9753.048} C_VEL
LIN {X 0,Y 425.282,Z 495.509,A -85,B 0,C 180,E1 -9755.928,E2 -9755.928} C_VEL
LIN {X 0,Y 425.277,Z 495.511,A -85,B 0,C 180,E1 -9759.04,E2 -9759.04} C_VEL
LIN {X 0,Y 425.291,Z 495.51,A -85,B 0,C 180,E1 -9761.958,E2 -9761.958} C_VEL
LIN {X 0,Y 425.286,Z 495.507,A -85,B 0,C 180,E1 -9765.283,E2 -9765.283} C_VEL
LIN {X 0,Y 425.316,Z 495.688,A -85,B 0,C 180,E1 -9767.243,E2 -9767.243} C_VEL
LIN {X 0,Y 427.376,Z 506.058,A -85,B 0,C 180,E1 -9770.614,E2 -9770.614} C_VEL
LIN {X 0,Y 428.663,Z 512.618,A -85,B 0,C 180,E1 -9772.654,E2 -9772.654} C_VEL
LIN {X 0,Y 428.705,Z 516.664,A -85,B 0,C 180,E1 -9773.831,E2 -9773.831} C_VEL
LIN {X 0,Y 427.795,Z 528.603,A -85,B 0,C 180,E1 -9777.171,E2 -9777.171} C_VEL
LIN {X 0,Y 427.021,Z 540.535,A -85,B 0,C 180,E1 -9780.413,E2 -9780.413} C_VEL
LIN {X 0,Y 426.244,Z 554.436,A -85,B 0,C 180,E1 -9784.091,E2 -9784.091} C_VEL
LIN {X 0,Y 425.711,Z 566.288,A -85,B 0,C 180,E1 -9787.173,E2 -9787.173} C_VEL
LIN {X 0,Y 425.203,Z 580.077,A -85,B 0,C 180,E1 -9790.697,E2 -9790.697} C_VEL
LIN {X 0,Y 424.982,Z 589.411,A -85,B 0,C 180,E1 -9793.052,E2 -9793.052} C_VEL
LIN {X 0,Y 426.565,Z 605.388,A -85,B 0,C 180,E1 -9793.584,E2 -9793.584} C_VEL
LIN {X 0,Y 427.444,Z 618.273,A -85,B 0,C 180,E1 -9794.198,E2 -9794.198} C_VEL
LIN {X 0,Y 427.815,Z 623.729,A -85,B 0,C 180,E1 -9794.517,E2 -9794.517} C_VEL
LIN {X 0,Y 427.129,Z 635.976,A -85,B 0,C 180,E1 -9795.346,E2 -9795.346} C_VEL
LIN {X 0,Y 426.459,Z 647.022,A -85,B 0,C 180,E1 -9796.297,E2 -9796.297} C_VEL
LIN {X 0,Y 425.984,Z 655.473,A -85,B 0,C 180,E1 -9797.188,E2 -9797.188} C_VEL
LIN {X 0,Y 425.415,Z 664.484,A -85,B 0,C 180,E1 -9798.324,E2 -9798.324} C_VEL
LIN {X 0,Y 424.918,Z 673.688,A -85,B 0,C 180,E1 -9799.758,E2 -9799.758} C_VEL
LIN {X 0,Y 424.703,Z 681.135,A -85,B 0,C 180,E1 -9801.195,E2 -9801.195} C_VEL
LIN {X 0,Y 424.597,Z 686.183,A -85,B 0,C 180,E1 -9802.391,E2 -9802.391} C_VEL
LIN {X 0,Y 424.579,Z 690.52,A -85,B 0,C 180,E1 -9803.64,E2 -9803.64} C_VEL
LIN {X 0,Y 424.648,Z 694.823,A -85,B 0,C 180,E1 -9805.253,E2 -9805.253} C_VEL
LIN {X 0,Y 424.683,Z 696.74,A -85,B 0,C 180,E1 -9806.205,E2 -9806.205} C_VEL
LIN {X 0,Y 424.661,Z 698.179,A -85,B 0,C 180,E1 -9807.154,E2 -9807.154} C_VEL
LIN {X 0,Y 424.682,Z 699.18,A -85,B 0,C 180,E1 -9808.103,E2 -9808.103} C_VEL
LIN {X 0,Y 424.882,Z 699.979,A -85,B 0,C 180,E1 -9810,E2 -9810} C_VEL
LIN {X 0,Y 424.711,Z 699.691,A -85,B 0,C 180,E1 -9810.948,E2 -9810.948} C_VEL
LIN {X 0,Y 424.705,Z 699.002,A -85,B 0,C 180,E1 -9811.897,E2 -9811.897} C_VEL
LIN {X 0,Y 424.688,Z 697.9,A -85,B 0,C 180,E1 -9812.846,E2 -9812.846} C_VEL
LIN {X 0,Y 424.704,Z 695.427,A -85,B 0,C 180,E1 -9814.271,E2 -9814.271} C_VEL
LIN {X 0,Y 424.606,Z 691.902,A -85,B 0,C 180,E1 -9815.7,E2 -9815.7} C_VEL
LIN {X 0,Y 424.623,Z 687.445,A -85,B 0,C 180,E1 -9817.083,E2 -9817.083} C_VEL
LIN {X 0,Y 424.717,Z 681.409,A -85,B 0,C 180,E1 -9818.565,E2 -9818.565} C_VEL
LIN {X 0,Y 424.879,Z 674.13,A -85,B 0,C 180,E1 -9820.002,E2 -9820.002} C_VEL
LIN {X 0,Y 425.342,Z 665.105,A -85,B 0,C 180,E1 -9821.436,E2 -9821.436} C_VEL
LIN {X 0,Y 425.894,Z 656.276,A -85,B 0,C 180,E1 -9822.59,E2 -9822.59} C_VEL
LIN {X 0,Y 426.225,Z 648.333,A -85,B 0,C 180,E1 -9823.468,E2 -9823.468} C_VEL
LIN {X 0,Y 426.955,Z 636.543,A -85,B 0,C 180,E1 -9824.538,E2 -9824.538} C_VEL
LIN {X 0,Y 427.722,Z 625.069,A -85,B 0,C 180,E1 -9825.364,E2 -9825.364} C_VEL
LIN {X 0,Y 427.616,Z 620.112,A -85,B 0,C 180,E1 -9825.674,E2 -9825.674} C_VEL
LIN {X 0,Y 426.935,Z 609.478,A -85,B 0,C 180,E1 -9826.251,E2 -9826.251} C_VEL
LIN {X 0,Y 426.046,Z 596.542,A -85,B 0,C 180,E1 -9826.786,E2 -9826.786} C_VEL
LIN {X 0,Y 424.898,Z 586.041,A -85,B 0,C 180,E1 -9827.109,E2 -9827.109} C_VEL
LIN {X 0,Y 425.191,Z 573.016,A -85,B 0,C 180,E1 -9830.311,E2 -9830.311} C_VEL
LIN {X 0,Y 425.544,Z 559.809,A -85,B 0,C 180,E1 -9833.61,E2 -9833.61} C_VEL
LIN {X 0,Y 426.041,Z 547.559,A -85,B 0,C 180,E1 -9836.741,E2 -9836.741} C_VEL
LIN {X 0,Y 426.612,Z 534.585,A -85,B 0,C 180,E1 -9840.163,E2 -9840.163} C_VEL
LIN {X 0,Y 427.205,Z 524.345,A -85,B 0,C 180,E1 -9842.964,E2 -9842.964} C_VEL
LIN {X 0,Y 428.095,Z 512.2,A -85,B 0,C 180,E1 -9846.445,E2 -9846.445} C_VEL
LIN {X 0,Y 427.66,Z 507.459,A -85,B 0,C 180,E1 -9847.925,E2 -9847.925} C_VEL
LIN {X 0,Y 426.121,Z 499.386,A -85,B 0,C 180,E1 -9850.652,E2 -9850.652} C_VEL
LIN {X 0,Y 425.32,Z 495.508,A -85,B 0,C 180,E1 -9852.123,E2 -9852.123} C_VEL
LIN {X 0,Y 425.287,Z 495.515,A -85,B 0,C 180,E1 -9855.283,E2 -9855.283} C_VEL
LIN {X 0,Y 425.277,Z 495.514,A -85,B 0,C 180,E1 -9858.622,E2 -9858.622} C_VEL
LIN {X 0,Y 425.308,Z 495.51,A -85,B 0,C 180,E1 -9861.102,E2 -9861.102} C_VEL
LIN {X 0,Y 425.3,Z 495.51,A -85,B 0,C 180,E1 -9864.664,E2 -9864.664} C_VEL
LIN {X 0,Y 425.267,Z 495.51,A -85,B 0,C 180,E1 -9868.073,E2 -9868.073} C_VEL
LIN {X 0,Y 425.334,Z 495.504,A -85,B 0,C 180,E1 -9871.368,E2 -9871.368} C_VEL
LIN {X 0,Y 425.357,Z 495.498,A -85,B 0,C 180,E1 -9873.506,E2 -9873.506} C_VEL
LIN {X 0,Y 425.308,Z 495.505,A -85,B 0,C 180,E1 -9876.635,E2 -9876.635} C_VEL
LIN {X 0,Y 425.332,Z 495.504,A -85,B 0,C 180,E1 -9880.365,E2 -9880.365} C_VEL
LIN {X 0,Y 425.392,Z 495.499,A -85,B 0,C 180,E1 -9883.689,E2 -9883.689} C_VEL
LIN {X 0,Y 425.416,Z 495.493,A -85,B 0,C 180,E1 -9887.598,E2 -9887.598} C_VEL
LIN {X 0,Y 425.446,Z 495.487,A -85,B 0,C 180,E1 -9891.45,E2 -9891.45} C_VEL
LIN {X 0,Y 425.558,Z 495.476,A -85,B 0,C 180,E1 -9894.314,E2 -9894.314} C_VEL
LIN {X 0,Y 425.575,Z 495.474,A -85,B 0,C 180,E1 -9898.108,E2 -9898.108} C_VEL
LIN {X 0,Y 425.704,Z 495.459,A -85,B 0,C 180,E1 -9900,E2 -9900} C_VEL
LIN {X 0,Y 425.549,Z 495.479,A -85,B 0,C 180,E1 -9902.84,E2 -9902.84} C_VEL
LIN {X 0,Y 425.485,Z 495.483,A -85,B 0,C 180,E1 -9906.543,E2 -9906.543} C_VEL
LIN {X 0,Y 425.404,Z 495.495,A -85,B 0,C 180,E1 -9909.51,E2 -9909.51} C_VEL
LIN {X 0,Y 425.398,Z 495.497,A -85,B 0,C 180,E1 -9912.904,E2 -9912.904} C_VEL
LIN {X 0,Y 425.377,Z 495.503,A -85,B 0,C 180,E1 -9916.61,E2 -9916.61} C_VEL
LIN {X 0,Y 425.362,Z 495.507,A -85,B 0,C 180,E1 -9917.767,E2 -9917.767} C_VEL
LIN {X 0,Y 428.89,Z 506.988,A -85,B 0,C 180,E1 -9918.635,E2 -9918.635} C_VEL
LIN {X 0,Y 429.602,Z 509.558,A -85,B 0,C 180,E1 -9918.851,E2 -9918.851} C_VEL
LIN {X 0,Y 429.166,Z 520.838,A -85,B 0,C 180,E1 -9919.741,E2 -9919.741} C_VEL
LIN {X 0,Y 428.548,Z 531.621,A -85,B 0,C 180,E1 -9920.807,E2 -9920.807} C_VEL
LIN {X 0,Y 427.891,Z 540.852,A -85,B 0,C 180,E1 -9921.942,E2 -9921.942} C_VEL
LIN {X 0,Y 427.276,Z 549.496,A -85,B 0,C 180,E1 -9923.252,E2 -9923.252} C_VEL
LIN {X 0,Y 426.717,Z 557.051,A -85,B 0,C 180,E1 -9924.668,E2 -9924.668} C_VEL
LIN {X 0,Y 426.237,Z 563.374,A -85,B 0,C 180,E1 -9926.172,E2 -9926.172} C_VEL
LIN {X 0,Y 425.881,Z 567.862,A -85,B 0,C 180,E1 -9927.521,E2 -9927.521} C_VEL
LIN {X 0,Y 425.599,Z 571.485,A -85,B 0,C 180,E1 -9928.931,E2 -9928.931} C_VEL
LIN {X 0,Y 425.283,Z 574.716,A -85,B 0,C 180,E1 -9930.758,E2 -9930.758} C_VEL
LIN {X 0,Y 425.108,Z 576.407,A -85,B 0,C 180,E1 -9932.525,E2 -9932.525} C_VEL
LIN {X 0,Y 425.051,Z 576.698,A -85,B 0,C 180,E1 -9934.236,E2 -9934.236} C_VEL
LIN {X 0,Y 425.055,Z 575.785,A -85,B 0,C 180,E1 -9935.886,E2 -9935.886} C_VEL
LIN {X 0,Y 425.192,Z 573.402,A -85,B 0,C 180,E1 -9937.704,E2 -9937.704} C_VEL
LIN {X 0,Y 425.433,Z 569.414,A -85,B 0,C 180,E1 -9939.53,E2 -9939.53} C_VEL
LIN {X 0,Y 425.701,Z 565.305,A -85,B 0,C 180,E1 -9940.902,E2 -9940.902} C_VEL
LIN {X 0,Y 426.118,Z 558.93,A -85,B 0,C 180,E1 -9942.549,E2 -9942.549} C_VEL
LIN {X 0,Y 426.502,Z 552.878,A -85,B 0,C 180,E1 -9943.796,E2 -9943.796} C_VEL
LIN {X 0,Y 427.088,Z 544.468,A -85,B 0,C 180,E1 -9945.207,E2 -9945.207} C_VEL
LIN {X 0,Y 427.64,Z 535.175,A -85,B 0,C 180,E1 -9946.466,E2 -9946.466} C_VEL
LIN {X 0,Y 428.221,Z 524.793,A -85,B 0,C 180,E1 -9947.608,E2 -9947.608} C_VEL
LIN {X 0,Y 428.786,Z 513.708,A -85,B 0,C 180,E1 -9948.581,E2 -9948.581} C_VEL
LIN {X 0,Y 428.97,Z 509.363,A -85,B 0,C 180,E1 -9948.907,E2 -9948.907} C_VEL
LIN {X 0,Y 427.074,Z 501.715,A -85,B 0,C 180,E1 -9949.498,E2 -9949.498} C_VEL
LIN {X 0,Y 425.299,Z 495.509,A -85,B 0,C 180,E1 -9949.947,E2 -9949.947} C_VEL
LIN {X 0,Y 425.268,Z 495.513,A -85,B 0,C 180,E1 -9953.491,E2 -9953.491} C_VEL
LIN {X 0,Y 425.312,Z 495.506,A -85,B 0,C 180,E1 -9955.817,E2 -9955.817} C_VEL
LIN {X 0,Y 425.296,Z 495.509,A -85,B 0,C 180,E1 -9959.239,E2 -9959.239} C_VEL
LIN {X 0,Y 425.351,Z 495.5,A -85,B 0,C 180,E1 -9962.442,E2 -9962.442} C_VEL
LIN {X 0,Y 425.351,Z 495.504,A -85,B 0,C 180,E1 -9965.602,E2 -9965.602} C_VEL
LIN {X 0,Y 425.299,Z 495.507,A -85,B 0,C 180,E1 -9968.682,E2 -9968.682} C_VEL
LIN {X 0,Y 425.327,Z 495.507,A -85,B 0,C 180,E1 -9971.702,E2 -9971.702} C_VEL
LIN {X 0,Y 425.352,Z 495.501,A -85,B 0,C 180,E1 -9974.671,E2 -9974.671} C_VEL
LIN {X 0,Y 425.418,Z 495.496,A -85,B 0,C 180,E1 -9977.598,E2 -9977.598} C_VEL
LIN {X 0,Y 425.414,Z 495.495,A -85,B 0,C 180,E1 -9981.449,E2 -9981.449} C_VEL
LIN {X 0,Y 425.538,Z 495.477,A -85,B 0,C 180,E1 -9984.313,E2 -9984.313} C_VEL
LIN {X 0,Y 425.578,Z 495.473,A -85,B 0,C 180,E1 -9988.107,E2 -9988.107} C_VEL
LIN {X 0,Y 425.698,Z 495.458,A -85,B 0,C 180,E1 -9990,E2 -9990} C_VEL
LIN {X 0,Y 425.541,Z 495.476,A -85,B 0,C 180,E1 -9992.516,E2 -9992.516} C_VEL
LIN {X 0,Y 424.865,Z 495.564,A -85,B 0,C 180,E1 -9993.305,E2 -9993.305} C_VEL
LIN {X 0,Y 421.989,Z 495.921,A -85,B 0,C 180,E1 -9994.587,E2 -9994.587} C_VEL
LIN {X 0,Y 419.562,Z 496.224,A -85,B 0,C 180,E1 -9995.621,E2 -9995.621} C_VEL
LIN {X 0,Y 418.528,Z 496.35,A -85,B 0,C 180,E1 -9996.421,E2 -9996.421} C_VEL
LIN {X 0,Y 418.448,Z 496.361,A -85,B 0,C 180,E1 -9996.692,E2 -9996.692} C_VEL
LIN {X 0,Y 418.344,Z 496.375,A -85,B 0,C 180,E1 -9999.671,E2 -9999.671} C_VEL
LIN {X 0,Y 418.352,Z 496.374,A -85,B 0,C 180,E1 -10003.001,E2 -10003.001} C_VEL
LIN {X 0,Y 418.317,Z 496.379,A -85,B 0,C 180,E1 -10006.735,E2 -10006.735} C_VEL
LIN {X 0,Y 418.275,Z 496.382,A -85,B 0,C 180,E1 -10009.79,E2 -10009.79} C_VEL
LIN {X 0,Y 418.242,Z 496.389,A -85,B 0,C 180,E1 -10012.736,E2 -10012.736} C_VEL
LIN {X 0,Y 418.241,Z 496.386,A -85,B 0,C 180,E1 -10015.906,E2 -10015.906} C_VEL
LIN {X 0,Y 418.265,Z 496.385,A -85,B 0,C 180,E1 -10019.162,E2 -10019.162} C_VEL
LIN {X 0,Y 418.261,Z 496.386,A -85,B 0,C 180,E1 -10022.844,E2 -10022.844} C_VEL
LIN {X 0,Y 418.247,Z 496.385,A -85,B 0,C 180,E1 -10026.237,E2 -10026.237} C_VEL
LIN {X 0,Y 418.213,Z 496.391,A -85,B 0,C 180,E1 -10029.686,E2 -10029.686} C_VEL
LIN {X 0,Y 418.215,Z 496.389,A -85,B 0,C 180,E1 -10032.318,E2 -10032.318} C_VEL
LIN {X 0,Y 418.239,Z 496.389,A -85,B 0,C 180,E1 -10035.108,E2 -10035.108} C_VEL
LIN {X 0,Y 418.237,Z 496.387,A -85,B 0,C 180,E1 -10037.766,E2 -10037.766} C_VEL
LIN {X 0,Y 418.245,Z 496.387,A -85,B 0,C 180,E1 -10040.621,E2 -10040.621} C_VEL
LIN {X 0,Y 418.245,Z 496.386,A -85,B 0,C 180,E1 -10043.975,E2 -10043.975} C_VEL
LIN {X 0,Y 418.261,Z 496.386,A -85,B 0,C 180,E1 -10047.156,E2 -10047.156} C_VEL
LIN {X 0,Y 418.272,Z 496.385,A -85,B 0,C 180,E1 -10050.895,E2 -10050.895} C_VEL
LIN {X 0,Y 418.264,Z 496.384,A -85,B 0,C 180,E1 -10054.095,E2 -10054.095} C_VEL
LIN {X 0,Y 418.234,Z 496.389,A -85,B 0,C 180,E1 -10057.263,E2 -10057.263} C_VEL
LIN {X 0,Y 418.286,Z 496.382,A -85,B 0,C 180,E1 -10060.364,E2 -10060.364} C_VEL
LIN {X 0,Y 418.319,Z 496.377,A -85,B 0,C 180,E1 -10063.404,E2 -10063.404} C_VEL
LIN {X 0,Y 418.349,Z 496.375,A -85,B 0,C 180,E1 -10066.999,E2 -10066.999} C_VEL
LIN {X 0,Y 418.341,Z 496.373,A -85,B 0,C 180,E1 -10070.328,E2 -10070.328} C_VEL
LIN {X 0,Y 418.461,Z 496.362,A -85,B 0,C 180,E1 -10073.248,E2 -10073.248} C_VEL
LIN {X 0,Y 418.337,Z 496.377,A -85,B 0,C 180,E1 -10075.181,E2 -10075.181} C_VEL
LIN {X 0,Y 418.542,Z 496.349,A -85,B 0,C 180,E1 -10078.075,E2 -10078.075} C_VEL
LIN {X 0,Y 418.669,Z 496.333,A -85,B 0,C 180,E1 -10080,E2 -10080} C_VEL
LIN {X 0,Y 418.489,Z 496.358,A -85,B 0,C 180,E1 -10082.888,E2 -10082.888} C_VEL
LIN {X 0,Y 418.492,Z 496.355,A -85,B 0,C 180,E1 -10085.783,E2 -10085.783} C_VEL
LIN {X 0,Y 418.398,Z 496.37,A -85,B 0,C 180,E1 -10088.695,E2 -10088.695} C_VEL
LIN {X 0,Y 418.332,Z 496.375,A -85,B 0,C 180,E1 -10091.63,E2 -10091.63} C_VEL
LIN {X 0,Y 418.307,Z 496.381,A -85,B 0,C 180,E1 -10094.597,E2 -10094.597} C_VEL
LIN {X 0,Y 418.281,Z 496.382,A -85,B 0,C 180,E1 -10097.604,E2 -10097.604} C_VEL
LIN {X 0,Y 418.252,Z 496.389,A -85,B 0,C 180,E1 -10100.663,E2 -10100.663} C_VEL
LIN {X 0,Y 418.287,Z 496.38,A -85,B 0,C 180,E1 -10103.781,E2 -10103.781} C_VEL
LIN {X 0,Y 418.228,Z 496.39,A -85,B 0,C 180,E1 -10107.048,E2 -10107.048} C_VEL
LIN {X 0,Y 418.243,Z 496.387,A -85,B 0,C 180,E1 -10110.272,E2 -10110.272} C_VEL
LIN {X 0,Y 418.248,Z 496.385,A -85,B 0,C 180,E1 -10113.677,E2 -10113.677} C_VEL
LIN {X 0,Y 418.24,Z 496.387,A -85,B 0,C 180,E1 -10117.224,E2 -10117.224} C_VEL
LIN {X 0,Y 418.244,Z 496.388,A -85,B 0,C 180,E1 -10119.683,E2 -10119.683} C_VEL
LIN {X 0,Y 418.231,Z 496.389,A -85,B 0,C 180,E1 -10122.321,E2 -10122.321} C_VEL
LIN {X 0,Y 418.236,Z 496.385,A -85,B 0,C 180,E1 -10125.109,E2 -10125.109} C_VEL
LIN {X 0,Y 418.281,Z 496.579,A -85,B 0,C 180,E1 -10126.93,E2 -10126.93} C_VEL
LIN {X 0,Y 420.304,Z 506.689,A -85,B 0,C 180,E1 -10130.28,E2 -10130.28} C_VEL
LIN {X 0,Y 421.677,Z 513.779,A -85,B 0,C 180,E1 -10132.531,E2 -10132.531} C_VEL
LIN {X 0,Y 421.755,Z 517.808,A -85,B 0,C 180,E1 -10133.732,E2 -10133.732} C_VEL
LIN {X 0,Y 420.786,Z 529.796,A -85,B 0,C 180,E1 -10137.141,E2 -10137.141} C_VEL
LIN {X 0,Y 420.035,Z 540.95,A -85,B 0,C 180,E1 -10140.229,E2 -10140.229} C_VEL
LIN {X 0,Y 419.158,Z 555.482,A -85,B 0,C 180,E1 -10144.155,E2 -10144.155} C_VEL
LIN {X 0,Y 418.568,Z 567.943,A -85,B 0,C 180,E1 -10147.441,E2 -10147.441} C_VEL
LIN {X 0,Y 418.084,Z 581.048,A -85,B 0,C 180,E1 -10150.865,E2 -10150.865} C_VEL
LIN {X 0,Y 417.92,Z 588.522,A -85,B 0,C 180,E1 -10152.794,E2 -10152.794} C_VEL
LIN {X 0,Y 419.435,Z 603.429,A -85,B 0,C 180,E1 -10153.284,E2 -10153.284} C_VEL
LIN {X 0,Y 420.244,Z 615.784,A -85,B 0,C 180,E1 -10153.857,E2 -10153.857} C_VEL
LIN {X 0,Y 420.829,Z 624.426,A -85,B 0,C 180,E1 -10154.378,E2 -10154.378} C_VEL
LIN {X 0,Y 420.111,Z 636.324,A -85,B 0,C 180,E1 -10155.22,E2 -10155.22} C_VEL
LIN {X 0,Y 419.423,Z 647.044,A -85,B 0,C 180,E1 -10156.186,E2 -10156.186} C_VEL
LIN {X 0,Y 418.924,Z 654.925,A -85,B 0,C 180,E1 -10157.039,E2 -10157.039} C_VEL
LIN {X 0,Y 418.326,Z 665.025,A -85,B 0,C 180,E1 -10158.369,E2 -10158.369} C_VEL
LIN {X 0,Y 417.824,Z 673.966,A -85,B 0,C 180,E1 -10159.827,E2 -10159.827} C_VEL
LIN {X 0,Y 417.626,Z 681.16,A -85,B 0,C 180,E1 -10161.289,E2 -10161.289} C_VEL
LIN {X 0,Y 417.487,Z 686.894,A -85,B 0,C 180,E1 -10162.747,E2 -10162.747} C_VEL
LIN {X 0,Y 417.501,Z 691.403,A -85,B 0,C 180,E1 -10164.203,E2 -10164.203} C_VEL
LIN {X 0,Y 417.602,Z 693.782,A -85,B 0,C 180,E1 -10165.173,E2 -10165.173} C_VEL
LIN {X 0,Y 417.646,Z 695.704,A -85,B 0,C 180,E1 -10166.141,E2 -10166.141} C_VEL
LIN {X 0,Y 417.621,Z 697.151,A -85,B 0,C 180,E1 -10167.106,E2 -10167.106} C_VEL
LIN {X 0,Y 417.647,Z 698.155,A -85,B 0,C 180,E1 -10168.071,E2 -10168.071} C_VEL
LIN {X 0,Y 417.861,Z 698.956,A -85,B 0,C 180,E1 -10170,E2 -10170} C_VEL
LIN {X 0,Y 417.681,Z 698.671,A -85,B 0,C 180,E1 -10170.964,E2 -10170.964} C_VEL
LIN {X 0,Y 417.669,Z 697.978,A -85,B 0,C 180,E1 -10171.929,E2 -10171.929} C_VEL
LIN {X 0,Y 417.647,Z 696.871,A -85,B 0,C 180,E1 -10172.894,E2 -10172.894} C_VEL
LIN {X 0,Y 417.673,Z 694.395,A -85,B 0,C 180,E1 -10174.343,E2 -10174.343} C_VEL
LIN {X 0,Y 417.55,Z 690.86,A -85,B 0,C 180,E1 -10175.796,E2 -10175.796} C_VEL
LIN {X 0,Y 417.559,Z 686.222,A -85,B 0,C 180,E1 -10177.252,E2 -10177.252} C_VEL
LIN {X 0,Y 417.655,Z 680.363,A -85,B 0,C 180,E1 -10178.711,E2 -10178.711} C_VEL
LIN {X 0,Y 417.828,Z 673.097,A -85,B 0,C 180,E1 -10180.173,E2 -10180.173} C_VEL
LIN {X 0,Y 418.307,Z 664.099,A -85,B 0,C 180,E1 -10181.631,E2 -10181.631} C_VEL
LIN {X 0,Y 418.863,Z 654.116,A -85,B 0,C 180,E1 -10182.945,E2 -10182.945} C_VEL
LIN {X 0,Y 419.543,Z 643.762,A -85,B 0,C 180,E1 -10184.058,E2 -10184.058} C_VEL
LIN {X 0,Y 420.309,Z 632.613,A -85,B 0,C 180,E1 -10185.021,E2 -10185.021} C_VEL
LIN {X 0,Y 420.81,Z 622.258,A -85,B 0,C 180,E1 -10185.747,E2 -10185.747} C_VEL
LIN {X 0,Y 420.138,Z 612.551,A -85,B 0,C 180,E1 -10186.334,E2 -10186.334} C_VEL
LIN {X 0,Y 419.344,Z 598.815,A -85,B 0,C 180,E1 -10186.965,E2 -10186.965} C_VEL
LIN {X 0,Y 417.852,Z 584.788,A -85,B 0,C 180,E1 -10187.45,E2 -10187.45} C_VEL
LIN {X 0,Y 418.128,Z 571.971,A -85,B 0,C 180,E1 -10190.67,E2 -10190.67} C_VEL
LIN {X 0,Y 418.56,Z 558.829,A -85,B 0,C 180,E1 -10194.028,E2 -10194.028} C_VEL
LIN {X 0,Y 419.006,Z 547.741,A -85,B 0,C 180,E1 -10196.928,E2 -10196.928} C_VEL
LIN {X 0,Y 419.576,Z 535.735,A -85,B 0,C 180,E1 -10200.166,E2 -10200.166} C_VEL
LIN {X 0,Y 420.26,Z 524.668,A -85,B 0,C 180,E1 -10203.264,E2 -10203.264} C_VEL
LIN {X 0,Y 421.071,Z 514.403,A -85,B 0,C 180,E1 -10206.264,E2 -10206.264} C_VEL
LIN {X 0,Y 420.936,Z 510.291,A -85,B 0,C 180,E1 -10207.547,E2 -10207.547} C_VEL
LIN {X 0,Y 419.538,Z 502.571,A -85,B 0,C 180,E1 -10210.169,E2 -10210.169} C_VEL
LIN {X 0,Y 418.269,Z 496.387,A -85,B 0,C 180,E1 -10212.449,E2 -10212.449} C_VEL
LIN {X 0,Y 418.238,Z 496.394,A -85,B 0,C 180,E1 -10215.109,E2 -10215.109} C_VEL
LIN {X 0,Y 418.243,Z 496.392,A -85,B 0,C 180,E1 -10217.767,E2 -10217.767} C_VEL
LIN {X 0,Y 418.255,Z 496.387,A -85,B 0,C 180,E1 -10220.62,E2 -10220.62} C_VEL
LIN {X 0,Y 418.244,Z 496.387,A -85,B 0,C 180,E1 -10223.976,E2 -10223.976} C_VEL
LIN {X 0,Y 418.26,Z 496.387,A -85,B 0,C 180,E1 -10227.156,E2 -10227.156} C_VEL
LIN {X 0,Y 418.272,Z 496.38,A -85,B 0,C 180,E1 -10230.896,E2 -10230.896} C_VEL
LIN {X 0,Y 418.271,Z 496.382,A -85,B 0,C 180,E1 -10234.096,E2 -10234.096} C_VEL
LIN {X 0,Y 418.241,Z 496.387,A -85,B 0,C 180,E1 -10237.264,E2 -10237.264} C_VEL
LIN {X 0,Y 418.287,Z 496.382,A -85,B 0,C 180,E1 -10240.364,E2 -10240.364} C_VEL
LIN {X 0,Y 418.32,Z 496.379,A -85,B 0,C 180,E1 -10243.405,E2 -10243.405} C_VEL
LIN {X 0,Y 418.35,Z 496.375,A -85,B 0,C 180,E1 -10246.999,E2 -10246.999} C_VEL
LIN {X 0,Y 418.344,Z 496.375,A -85,B 0,C 180,E1 -10250.329,E2 -10250.329} C_VEL
LIN {X 0,Y 418.517,Z 496.35,A -85,B 0,C 180,E1 -10252.28,E2 -10252.28} C_VEL
LIN {X 0,Y 418.517,Z 496.353,A -85,B 0,C 180,E1 -10254.218,E2 -10254.218} C_VEL
LIN {X 0,Y 418.544,Z 496.349,A -85,B 0,C 180,E1 -10258.076,E2 -10258.076} C_VEL
LIN {X 0,Y 418.673,Z 496.334,A -85,B 0,C 180,E1 -10260,E2 -10260} C_VEL
LIN {X 0,Y 418.504,Z 496.356,A -85,B 0,C 180,E1 -10262.888,E2 -10262.888} C_VEL
LIN {X 0,Y 418.449,Z 496.359,A -85,B 0,C 180,E1 -10266.542,E2 -10266.542} C_VEL
LIN {X 0,Y 418.345,Z 496.376,A -85,B 0,C 180,E1 -10269.672,E2 -10269.672} C_VEL
LIN {X 0,Y 418.351,Z 496.374,A -85,B 0,C 180,E1 -10273.001,E2 -10273.001} C_VEL
LIN {X 0,Y 418.344,Z 496.379,A -85,B 0,C 180,E1 -10276.748,E2 -10276.748} C_VEL
LIN {X 0,Y 418.327,Z 496.485,A -85,B 0,C 180,E1 -10277.465,E2 -10277.465} C_VEL
LIN {X 0,Y 422.157,Z 508.562,A -85,B 0,C 180,E1 -10278.389,E2 -10278.389} C_VEL
LIN {X 0,Y 422.897,Z 513.059,A -85,B 0,C 180,E1 -10278.757,E2 -10278.757} C_VEL
LIN {X 0,Y 422.294,Z 524.265,A -85,B 0,C 180,E1 -10279.695,E2 -10279.695} C_VEL
LIN {X 0,Y 421.613,Z 534.978,A -85,B 0,C 180,E1 -10280.831,E2 -10280.831} C_VEL
LIN {X 0,Y 420.909,Z 544.393,A -85,B 0,C 180,E1 -10282.067,E2 -10282.067} C_VEL
LIN {X 0,Y 420.288,Z 552.245,A -85,B 0,C 180,E1 -10283.341,E2 -10283.341} C_VEL
LIN {X 0,Y 419.744,Z 559.246,A -85,B 0,C 180,E1 -10284.746,E2 -10284.746} C_VEL
LIN {X 0,Y 419.19,Z 565.703,A -85,B 0,C 180,E1 -10286.378,E2 -10286.378} C_VEL
LIN {X 0,Y 418.76,Z 570.67,A -85,B 0,C 180,E1 -10288.03,E2 -10288.03} C_VEL
LIN {X 0,Y 418.54,Z 573.252,A -85,B 0,C 180,E1 -10289.17,E2 -10289.17} C_VEL
LIN {X 0,Y 418.258,Z 576.197,A -85,B 0,C 180,E1 -10291.023,E2 -10291.023} C_VEL
LIN {X 0,Y 418.09,Z 577.577,A -85,B 0,C 180,E1 -10292.807,E2 -10292.807} C_VEL
LIN {X 0,Y 418.028,Z 577.648,A -85,B 0,C 180,E1 -10294.532,E2 -10294.532} C_VEL
LIN {X 0,Y 418.052,Z 576.526,A -85,B 0,C 180,E1 -10296.201,E2 -10296.201} C_VEL
LIN {X 0,Y 418.178,Z 574.281,A -85,B 0,C 180,E1 -10297.824,E2 -10297.824} C_VEL
LIN {X 0,Y 418.436,Z 570.253,A -85,B 0,C 180,E1 -10299.662,E2 -10299.662} C_VEL
LIN {X 0,Y 418.831,Z 564.501,A -85,B 0,C 180,E1 -10301.515,E2 -10301.515} C_VEL
LIN {X 0,Y 419.246,Z 557.762,A -85,B 0,C 180,E1 -10303.144,E2 -10303.144} C_VEL
LIN {X 0,Y 419.854,Z 549.76,A -85,B 0,C 180,E1 -10304.672,E2 -10304.672} C_VEL
LIN {X 0,Y 420.475,Z 540.26,A -85,B 0,C 180,E1 -10306.111,E2 -10306.111} C_VEL
LIN {X 0,Y 421.051,Z 530.922,A -85,B 0,C 180,E1 -10307.26,E2 -10307.26} C_VEL
LIN {X 0,Y 421.628,Z 520.277,A -85,B 0,C 180,E1 -10308.325,E2 -10308.325} C_VEL
LIN {X 0,Y 422.099,Z 511.143,A -85,B 0,C 180,E1 -10309.066,E2 -10309.066} C_VEL
LIN {X 0,Y 421.247,Z 506.906,A -85,B 0,C 180,E1 -10309.408,E2 -10309.408} C_VEL
LIN {X 0,Y 418.227,Z 496.39,A -85,B 0,C 180,E1 -10310.198,E2 -10310.198} C_VEL
LIN {X 0,Y 418.243,Z 496.389,A -85,B 0,C 180,E1 -10312.776,E2 -10312.776} C_VEL
LIN {X 0,Y 418.254,Z 496.384,A -85,B 0,C 180,E1 -10316.323,E2 -10316.323} C_VEL
LIN {X 0,Y 418.25,Z 496.388,A -85,B 0,C 180,E1 -10319.728,E2 -10319.728} C_VEL
LIN {X 0,Y 418.31,Z 496.38,A -85,B 0,C 180,E1 -10323.023,E2 -10323.023} C_VEL
LIN {X 0,Y 418.279,Z 496.381,A -85,B 0,C 180,E1 -10326.218,E2 -10326.218} C_VEL
LIN {X 0,Y 418.255,Z 496.387,A -85,B 0,C 180,E1 -10329.337,E2 -10329.337} C_VEL
LIN {X 0,Y 418.285,Z 496.38,A -85,B 0,C 180,E1 -10332.396,E2 -10332.396} C_VEL
LIN {X 0,Y 418.307,Z 496.38,A -85,B 0,C 180,E1 -10335.403,E2 -10335.403} C_VEL
LIN {X 0,Y 418.321,Z 496.376,A -85,B 0,C 180,E1 -10338.369,E2 -10338.369} C_VEL
LIN {X 0,Y 418.383,Z 496.371,A -85,B 0,C 180,E1 -10341.304,E2 -10341.304} C_VEL
LIN {X 0,Y 418.495,Z 496.354,A -85,B 0,C 180,E1 -10344.217,E2 -10344.217} C_VEL
LIN {X 0,Y 418.547,Z 496.349,A -85,B 0,C 180,E1 -10348.075,E2 -10348.075} C_VEL
LIN {X 0,Y 418.667,Z 496.333,A -85,B 0,C 180,E1 -10350,E2 -10350} C_VEL
LIN {X 0,Y 418.498,Z 496.356,A -85,B 0,C 180,E1 -10352.888,E2 -10352.888} C_VEL
LIN {X 0,Y 418.494,Z 496.356,A -85,B 0,C 180,E1 -10355.783,E2 -10355.783} C_VEL
LIN {X 0,Y 418.448,Z 496.361,A -85,B 0,C 180,E1 -10356.692,E2 -10356.692} C_VEL
LIN {X 0,Y 417.786,Z 496.448,A -85,B 0,C 180,E1 -10357.494,E2 -10357.494} C_VEL
LIN {X 0,Y 414.906,Z 496.811,A -85,B 0,C 180,E1 -10358.797,E2 -10358.797} C_VEL
LIN {X 0,Y 412.45,Z 497.116,A -85,B 0,C 180,E1 -10359.849,E2 -10359.849} C_VEL
LIN {X 0,Y 411.38,Z 497.245,A -85,B 0,C 180,E1 -10360.663,E2 -10360.663} C_VEL
LIN {X 0,Y 411.284,Z 497.254,A -85,B 0,C 180,E1 -10360.939,E2 -10360.939} C_VEL
LIN {X 0,Y 411.26,Z 497.256,A -85,B 0,C 180,E1 -10363.842,E2 -10363.842} C_VEL
LIN {X 0,Y 411.262,Z 497.258,A -85,B 0,C 180,E1 -10366.888,E2 -10366.888} C_VEL
LIN {X 0,Y 411.235,Z 497.258,A -85,B 0,C 180,E1 -10369.987,E2 -10369.987} C_VEL
LIN {X 0,Y 411.206,Z 497.265,A -85,B 0,C 180,E1 -10373.147,E2 -10373.147} C_VEL
LIN {X 0,Y 411.207,Z 497.262,A -85,B 0,C 180,E1 -10376.383,E2 -10376.383} C_VEL
LIN {X 0,Y 411.202,Z 497.264,A -85,B 0,C 180,E1 -10379.713,E2 -10379.713} C_VEL
LIN {X 0,Y 411.21,Z 497.265,A -85,B 0,C 180,E1 -10383.155,E2 -10383.155} C_VEL
LIN {X 0,Y 411.195,Z 497.264,A -85,B 0,C 180,E1 -10386.552,E2 -10386.552} C_VEL
LIN {X 0,Y 411.181,Z 497.267,A -85,B 0,C 180,E1 -10389.722,E2 -10389.722} C_VEL
LIN {X 0,Y 411.168,Z 497.271,A -85,B 0,C 180,E1 -10393.134,E2 -10393.134} C_VEL
LIN {X 0,Y 411.17,Z 497.267,A -85,B 0,C 180,E1 -10395.881,E2 -10395.881} C_VEL
LIN {X 0,Y 411.163,Z 497.269,A -85,B 0,C 180,E1 -10398.772,E2 -10398.772} C_VEL
LIN {X 0,Y 411.192,Z 497.264,A -85,B 0,C 180,E1 -10402.025,E2 -10402.025} C_VEL
LIN {X 0,Y 411.209,Z 497.262,A -85,B 0,C 180,E1 -10405.666,E2 -10405.666} C_VEL
LIN {X 0,Y 411.193,Z 497.267,A -85,B 0,C 180,E1 -10409.152,E2 -10409.152} C_VEL
LIN {X 0,Y 411.262,Z 497.256,A -85,B 0,C 180,E1 -10412.522,E2 -10412.522} C_VEL
LIN {X 0,Y 411.214,Z 497.262,A -85,B 0,C 180,E1 -10415.783,E2 -10415.783} C_VEL
LIN {X 0,Y 411.199,Z 497.267,A -85,B 0,C 180,E1 -10418.966,E2 -10418.966} C_VEL
LIN {X 0,Y 411.253,Z 497.256,A -85,B 0,C 180,E1 -10422.085,E2 -10422.085} C_VEL
LIN {X 0,Y 411.262,Z 497.258,A -85,B 0,C 180,E1 -10425.147,E2 -10425.147} C_VEL
LIN {X 0,Y 411.286,Z 497.253,A -85,B 0,C 180,E1 -10428.167,E2 -10428.167} C_VEL
LIN {X 0,Y 411.321,Z 497.25,A -85,B 0,C 180,E1 -10431.154,E2 -10431.154} C_VEL
LIN {X 0,Y 411.444,Z 497.233,A -85,B 0,C 180,E1 -10434.117,E2 -10434.117} C_VEL
LIN {X 0,Y 411.511,Z 497.225,A -85,B 0,C 180,E1 -10438.042,E2 -10438.042} C_VEL
LIN {X 0,Y 411.638,Z 497.208,A -85,B 0,C 180,E1 -10440,E2 -10440} C_VEL
LIN {X 0,Y 411.445,Z 497.235,A -85,B 0,C 180,E1 -10442.937,E2 -10442.937} C_VEL
LIN {X 0,Y 411.436,Z 497.234,A -85,B 0,C 180,E1 -10445.882,E2 -10445.882} C_VEL
LIN {X 0,Y 411.354,Z 497.247,A -85,B 0,C 180,E1 -10448.845,E2 -10448.845} C_VEL
LIN {X 0,Y 411.3,Z 497.251,A -85,B 0,C 180,E1 -10451.832,E2 -10451.832} C_VEL
LIN {X 0,Y 411.263,Z 497.258,A -85,B 0,C 180,E1 -10454.852,E2 -10454.852} C_VEL
LIN {X 0,Y 411.247,Z 497.257,A -85,B 0,C 180,E1 -10457.915,E2 -10457.915} C_VEL
LIN {X 0,Y 411.198,Z 497.265,A -85,B 0,C 180,E1 -10461.034,E2 -10461.034} C_VEL
LIN {X 0,Y 411.219,Z 497.262,A -85,B 0,C 180,E1 -10464.216,E2 -10464.216} C_VEL
LIN {X 0,Y 411.189,Z 497.265,A -85,B 0,C 180,E1 -10467.483,E2 -10467.483} C_VEL
LIN {X 0,Y 411.19,Z 497.268,A -85,B 0,C 180,E1 -10470.847,E2 -10470.847} C_VEL
LIN {X 0,Y 411.206,Z 497.265,A -85,B 0,C 180,E1 -10474.333,E2 -10474.333} C_VEL
LIN {X 0,Y 411.191,Z 497.263,A -85,B 0,C 180,E1 -10477.974,E2 -10477.974} C_VEL
LIN {X 0,Y 411.165,Z 497.271,A -85,B 0,C 180,E1 -10481.228,E2 -10481.228} C_VEL
LIN {X 0,Y 411.177,Z 497.266,A -85,B 0,C 180,E1 -10484.49,E2 -10484.49} C_VEL
LIN {X 0,Y 411.211,Z 497.441,A -85,B 0,C 180,E1 -10486.593,E2 -10486.593} C_VEL
LIN {X 0,Y 413.195,Z 507.311,A -85,B 0,C 180,E1 -10489.943,E2 -10489.943} C_VEL
LIN {X 0,Y 414.83,Z 516.117,A -85,B 0,C 180,E1 -10492.775,E2 -10492.775} C_VEL
LIN {X 0,Y 414.537,Z 521.812,A -85,B 0,C 180,E1 -10494.467,E2 -10494.467} C_VEL
LIN {X 0,Y 413.646,Z 532.842,A -85,B 0,C 180,E1 -10497.643,E2 -10497.643} C_VEL
LIN {X 0,Y 412.935,Z 542.719,A -85,B 0,C 180,E1 -10500.425,E2 -10500.425} C_VEL
LIN {X 0,Y 412.086,Z 556.543,A -85,B 0,C 180,E1 -10504.222,E2 -10504.222} C_VEL
LIN {X 0,Y 411.46,Z 569.001,A -85,B 0,C 180,E1 -10507.586,E2 -10507.586} C_VEL
LIN {X 0,Y 410.983,Z 582.025,A -85,B 0,C 180,E1 -10511.04,E2 -10511.04} C_VEL
LIN {X 0,Y 410.837,Z 587.668,A -85,B 0,C 180,E1 -10512.526,E2 -10512.526} C_VEL
LIN {X 0,Y 412.325,Z 602.321,A -85,B 0,C 180,E1 -10513.013,E2 -10513.013} C_VEL
LIN {X 0,Y 413.209,Z 615.411,A -85,B 0,C 180,E1 -10513.639,E2 -10513.639} C_VEL
LIN {X 0,Y 413.837,Z 624.988,A -85,B 0,C 180,E1 -10514.233,E2 -10514.233} C_VEL
LIN {X 0,Y 413.094,Z 636.489,A -85,B 0,C 180,E1 -10515.089,E2 -10515.089} C_VEL
LIN {X 0,Y 412.39,Z 646.999,A -85,B 0,C 180,E1 -10516.071,E2 -10516.071} C_VEL
LIN {X 0,Y 411.848,Z 654.309,A -85,B 0,C 180,E1 -10516.883,E2 -10516.883} C_VEL
LIN {X 0,Y 411.329,Z 662.202,A -85,B 0,C 180,E1 -10517.918,E2 -10517.918} C_VEL
LIN {X 0,Y 410.853,Z 671.478,A -85,B 0,C 180,E1 -10519.404,E2 -10519.404} C_VEL
LIN {X 0,Y 410.559,Z 678.961,A -85,B 0,C 180,E1 -10520.889,E2 -10520.889} C_VEL
LIN {X 0,Y 410.458,Z 684.046,A -85,B 0,C 180,E1 -10522.127,E2 -10522.127} C_VEL
LIN {X 0,Y 410.465,Z 688.952,A -85,B 0,C 180,E1 -10523.603,E2 -10523.603} C_VEL
LIN {X 0,Y 410.556,Z 692.74,A -85,B 0,C 180,E1 -10525.09,E2 -10525.09} C_VEL
LIN {X 0,Y 410.61,Z 694.668,A -85,B 0,C 180,E1 -10526.074,E2 -10526.074} C_VEL
LIN {X 0,Y 410.582,Z 696.123,A -85,B 0,C 180,E1 -10527.057,E2 -10527.057} C_VEL
LIN {X 0,Y 410.611,Z 697.127,A -85,B 0,C 180,E1 -10528.038,E2 -10528.038} C_VEL
LIN {X 0,Y 410.84,Z 697.933,A -85,B 0,C 180,E1 -10530,E2 -10530} C_VEL
LIN {X 0,Y 410.651,Z 697.65,A -85,B 0,C 180,E1 -10530.981,E2 -10530.981} C_VEL
LIN {X 0,Y 410.632,Z 696.952,A -85,B 0,C 180,E1 -10531.962,E2 -10531.962} C_VEL
LIN {X 0,Y 410.606,Z 695.844,A -85,B 0,C 180,E1 -10532.943,E2 -10532.943} C_VEL
LIN {X 0,Y 410.623,Z 693.367,A -85,B 0,C 180,E1 -10534.417,E2 -10534.417} C_VEL
LIN {X 0,Y 410.486,Z 689.833,A -85,B 0,C 180,E1 -10535.896,E2 -10535.896} C_VEL
LIN {X 0,Y 410.479,Z 685.198,A -85,B 0,C 180,E1 -10537.378,E2 -10537.378} C_VEL
LIN {X 0,Y 410.571,Z 679.339,A -85,B 0,C 180,E1 -10538.862,E2 -10538.862} C_VEL
LIN {X 0,Y 410.772,Z 672.078,A -85,B 0,C 180,E1 -10540.349,E2 -10540.349} C_VEL
LIN {X 0,Y 411.195,Z 664.739,A -85,B 0,C 180,E1 -10541.585,E2 -10541.585} C_VEL
LIN {X 0,Y 411.783,Z 655.965,A -85,B 0,C 180,E1 -10542.819,E2 -10542.819} C_VEL
LIN {X 0,Y 412.198,Z 647.546,A -85,B 0,C 180,E1 -10543.81,E2 -10543.81} C_VEL
LIN {X 0,Y 413.029,Z 636.12,A -85,B 0,C 180,E1 -10544.914,E2 -10544.914} C_VEL
LIN {X 0,Y 413.836,Z 625.108,A -85,B 0,C 180,E1 -10545.767,E2 -10545.767} C_VEL
LIN {X 0,Y 413.245,Z 613.024,A -85,B 0,C 180,E1 -10546.551,E2 -10546.551} C_VEL
LIN {X 0,Y 412.55,Z 599.867,A -85,B 0,C 180,E1 -10547.204,E2 -10547.204} C_VEL
LIN {X 0,Y 411.182,Z 587.162,A -85,B 0,C 180,E1 -10547.674,E2 -10547.674} C_VEL
LIN {X 0,Y 410.807,Z 583.524,A -85,B 0,C 180,E1 -10547.813,E2 -10547.813} C_VEL
LIN {X 0,Y 411.09,Z 570.963,A -85,B 0,C 180,E1 -10551.04,E2 -10551.04} C_VEL
LIN {X 0,Y 411.502,Z 558.874,A -85,B 0,C 180,E1 -10554.198,E2 -10554.198} C_VEL
LIN {X 0,Y 411.938,Z 548.834,A -85,B 0,C 180,E1 -10556.88,E2 -10556.88} C_VEL
LIN {X 0,Y 412.536,Z 536.878,A -85,B 0,C 180,E1 -10560.17,E2 -10560.17} C_VEL
LIN {X 0,Y 413.267,Z 526.001,A -85,B 0,C 180,E1 -10563.276,E2 -10563.276} C_VEL
LIN {X 0,Y 414.139,Z 515.417,A -85,B 0,C 180,E1 -10566.439,E2 -10566.439} C_VEL
LIN {X 0,Y 413.97,Z 511.556,A -85,B 0,C 180,E1 -10567.675,E2 -10567.675} C_VEL
LIN {X 0,Y 412.301,Z 502.489,A -85,B 0,C 180,E1 -10570.856,E2 -10570.856} C_VEL
LIN {X 0,Y 411.2,Z 497.269,A -85,B 0,C 180,E1 -10572.86,E2 -10572.86} C_VEL
LIN {X 0,Y 411.171,Z 497.274,A -85,B 0,C 180,E1 -10575.881,E2 -10575.881} C_VEL
LIN {X 0,Y 411.166,Z 497.272,A -85,B 0,C 180,E1 -10578.772,E2 -10578.772} C_VEL
LIN {X 0,Y 411.206,Z 497.262,A -85,B 0,C 180,E1 -10581.832,E2 -10581.832} C_VEL
LIN {X 0,Y 411.212,Z 497.264,A -85,B 0,C 180,E1 -10585.122,E2 -10585.122} C_VEL
LIN {X 0,Y 411.168,Z 497.266,A -85,B 0,C 180,E1 -10588.003,E2 -10588.003} C_VEL
LIN {X 0,Y 411.221,Z 497.262,A -85,B 0,C 180,E1 -10591.41,E2 -10591.41} C_VEL
LIN {X 0,Y 411.24,Z 497.256,A -85,B 0,C 180,E1 -10593.619,E2 -10593.619} C_VEL
LIN {X 0,Y 411.205,Z 497.262,A -85,B 0,C 180,E1 -10596.853,E2 -10596.853} C_VEL
LIN {X 0,Y 411.219,Z 497.263,A -85,B 0,C 180,E1 -10600.051,E2 -10600.051} C_VEL
LIN {X 0,Y 411.267,Z 497.256,A -85,B 0,C 180,E1 -10603.131,E2 -10603.131} C_VEL
LIN {X 0,Y 411.309,Z 497.252,A -85,B 0,C 180,E1 -10606.896,E2 -10606.896} C_VEL
LIN {X 0,Y 411.296,Z 497.254,A -85,B 0,C 180,E1 -10610.162,E2 -10610.162} C_VEL
LIN {X 0,Y 411.486,Z 497.225,A -85,B 0,C 180,E1 -10612.147,E2 -10612.147} C_VEL
LIN {X 0,Y 411.479,Z 497.23,A -85,B 0,C 180,E1 -10614.118,E2 -10614.118} C_VEL
LIN {X 0,Y 411.513,Z 497.225,A -85,B 0,C 180,E1 -10618.043,E2 -10618.043} C_VEL
LIN {X 0,Y 411.643,Z 497.21,A -85,B 0,C 180,E1 -10620,E2 -10620} C_VEL
LIN {X 0,Y 411.461,Z 497.234,A -85,B 0,C 180,E1 -10622.938,E2 -10622.938} C_VEL
LIN {X 0,Y 411.398,Z 497.237,A -85,B 0,C 180,E1 -10626.539,E2 -10626.539} C_VEL
LIN {X 0,Y 411.297,Z 497.256,A -85,B 0,C 180,E1 -10629.839,E2 -10629.839} C_VEL
LIN {X 0,Y 411.31,Z 497.251,A -85,B 0,C 180,E1 -10633.104,E2 -10633.104} C_VEL
LIN {X 0,Y 411.307,Z 497.257,A -85,B 0,C 180,E1 -10636.887,E2 -10636.887} C_VEL
LIN {X 0,Y 411.274,Z 497.262,A -85,B 0,C 180,E1 -10637.11,E2 -10637.11} C_VEL
LIN {X 0,Y 415.326,Z 509.93,A -85,B 0,C 180,E1 -10638.116,E2 -10638.116} C_VEL
LIN {X 0,Y 416.2,Z 513.875,A -85,B 0,C 180,E1 -10638.459,E2 -10638.459} C_VEL
LIN {X 0,Y 415.641,Z 524.407,A -85,B 0,C 180,E1 -10639.342,E2 -10639.342} C_VEL
LIN {X 0,Y 414.924,Z 534.91,A -85,B 0,C 180,E1 -10640.448,E2 -10640.448} C_VEL
LIN {X 0,Y 414.185,Z 544.482,A -85,B 0,C 180,E1 -10641.699,E2 -10641.699} C_VEL
LIN {X 0,Y 413.5,Z 552.641,A -85,B 0,C 180,E1 -10643.012,E2 -10643.012} C_VEL
LIN {X 0,Y 412.937,Z 559.513,A -85,B 0,C 180,E1 -10644.376,E2 -10644.376} C_VEL
LIN {X 0,Y 412.431,Z 565.361,A -85,B 0,C 180,E1 -10645.82,E2 -10645.82} C_VEL
LIN {X 0,Y 411.913,Z 570.585,A -85,B 0,C 180,E1 -10647.474,E2 -10647.474} C_VEL
LIN {X 0,Y 411.702,Z 573.262,A -85,B 0,C 180,E1 -10648.554,E2 -10648.554} C_VEL
LIN {X 0,Y 411.441,Z 575.457,A -85,B 0,C 180,E1 -10649.694,E2 -10649.694} C_VEL
LIN {X 0,Y 411.188,Z 577.589,A -85,B 0,C 180,E1 -10651.284,E2 -10651.284} C_VEL
LIN {X 0,Y 411.051,Z 578.764,A -85,B 0,C 180,E1 -10653.17,E2 -10653.17} C_VEL
LIN {X 0,Y 411,Z 578.572,A -85,B 0,C 180,E1 -10654.836,E2 -10654.836} C_VEL
LIN {X 0,Y 411.056,Z 576.917,A -85,B 0,C 180,E1 -10656.757,E2 -10656.757} C_VEL
LIN {X 0,Y 411.25,Z 573.819,A -85,B 0,C 180,E1 -10658.642,E2 -10658.642} C_VEL
LIN {X 0,Y 411.594,Z 569.25,A -85,B 0,C 180,E1 -10660.456,E2 -10660.456} C_VEL
LIN {X 0,Y 411.944,Z 564.059,A -85,B 0,C 180,E1 -10662.001,E2 -10662.001} C_VEL
LIN {X 0,Y 412.454,Z 557.03,A -85,B 0,C 180,E1 -10663.639,E2 -10663.639} C_VEL
LIN {X 0,Y 412.963,Z 550.105,A -85,B 0,C 180,E1 -10664.932,E2 -10664.932} C_VEL
LIN {X 0,Y 413.575,Z 541.118,A -85,B 0,C 180,E1 -10666.303,E2 -10666.303} C_VEL
LIN {X 0,Y 414.216,Z 531.221,A -85,B 0,C 180,E1 -10667.531,E2 -10667.531} C_VEL
LIN {X 0,Y 414.793,Z 521.089,A -85,B 0,C 180,E1 -10668.55,E2 -10668.55} C_VEL
LIN {X 0,Y 415.206,Z 511.608,A -85,B 0,C 180,E1 -10669.332,E2 -10669.332} C_VEL
LIN {X 0,Y 412.017,Z 500.233,A -85,B 0,C 180,E1 -10670.235,E2 -10670.235} C_VEL
LIN {X 0,Y 411.197,Z 497.266,A -85,B 0,C 180,E1 -10670.459,E2 -10670.459} C_VEL
LIN {X 0,Y 411.197,Z 497.266,A -85,B 0,C 180,E1 -10673.448,E2 -10673.448} C_VEL
LIN {X 0,Y 411.212,Z 497.262,A -85,B 0,C 180,E1 -10676.873,E2 -10676.873} C_VEL
LIN {X 0,Y 411.238,Z 497.258,A -85,B 0,C 180,E1 -10680.644,E2 -10680.644} C_VEL
LIN {X 0,Y 411.239,Z 497.26,A -85,B 0,C 180,E1 -10683.619,E2 -10683.619} C_VEL
LIN {X 0,Y 411.201,Z 497.264,A -85,B 0,C 180,E1 -10686.852,E2 -10686.852} C_VEL
LIN {X 0,Y 411.22,Z 497.262,A -85,B 0,C 180,E1 -10690.05,E2 -10690.05} C_VEL
LIN {X 0,Y 411.269,Z 497.257,A -85,B 0,C 180,E1 -10693.131,E2 -10693.131} C_VEL
LIN {X 0,Y 411.311,Z 497.252,A -85,B 0,C 180,E1 -10696.896,E2 -10696.896} C_VEL
LIN {X 0,Y 411.297,Z 497.25,A -85,B 0,C 180,E1 -10700.161,E2 -10700.161} C_VEL
LIN {X 0,Y 411.398,Z 497.241,A -85,B 0,C 180,E1 -10703.132,E2 -10703.132} C_VEL
LIN {X 0,Y 411.309,Z 497.252,A -85,B 0,C 180,E1 -10705.099,E2 -10705.099} C_VEL
LIN {X 0,Y 411.516,Z 497.224,A -85,B 0,C 180,E1 -10708.042,E2 -10708.042} C_VEL
LIN {X 0,Y 411.637,Z 497.209,A -85,B 0,C 180,E1 -10710,E2 -10710} C_VEL
LIN {X 0,Y 411.454,Z 497.234,A -85,B 0,C 180,E1 -10712.937,E2 -10712.937} C_VEL
LIN {X 0,Y 411.396,Z 497.239,A -85,B 0,C 180,E1 -10716.691,E2 -10716.691} C_VEL
LIN {X 0,Y 411.296,Z 497.253,A -85,B 0,C 180,E1 -10719.839,E2 -10719.839} C_VEL
LIN {X 0,Y 411.284,Z 497.254,A -85,B 0,C 180,E1 -10720.939,E2 -10720.939} C_VEL
LIN {X 0,Y 410.597,Z 497.34,A -85,B 0,C 180,E1 -10721.756,E2 -10721.756} C_VEL
LIN {X 0,Y 407.741,Z 497.697,A -85,B 0,C 180,E1 -10723.085,E2 -10723.085} C_VEL
LIN {X 0,Y 405.333,Z 498,A -85,B 0,C 180,E1 -10724.157,E2 -10724.157} C_VEL
LIN {X 0,Y 404.293,Z 498.128,A -85,B 0,C 180,E1 -10724.986,E2 -10724.986} C_VEL
LIN {X 0,Y 404.205,Z 498.136,A -85,B 0,C 180,E1 -10725.267,E2 -10725.267} C_VEL
LIN {X 0,Y 404.209,Z 498.133,A -85,B 0,C 180,E1 -10728.238,E2 -10728.238} C_VEL
LIN {X 0,Y 404.143,Z 498.144,A -85,B 0,C 180,E1 -10731.419,E2 -10731.419} C_VEL
LIN {X 0,Y 404.171,Z 498.14,A -85,B 0,C 180,E1 -10734.666,E2 -10734.666} C_VEL
LIN {X 0,Y 404.171,Z 498.139,A -85,B 0,C 180,E1 -10738.001,E2 -10738.001} C_VEL
LIN {X 0,Y 404.143,Z 498.143,A -85,B 0,C 180,E1 -10741.558,E2 -10741.558} C_VEL
LIN {X 0,Y 404.187,Z 498.139,A -85,B 0,C 180,E1 -10745.016,E2 -10745.016} C_VEL
LIN {X 0,Y 404.14,Z 498.144,A -85,B 0,C 180,E1 -10748.759,E2 -10748.759} C_VEL
LIN {X 0,Y 404.113,Z 498.147,A -85,B 0,C 180,E1 -10751.597,E2 -10751.597} C_VEL
LIN {X 0,Y 404.147,Z 498.142,A -85,B 0,C 180,E1 -10754.522,E2 -10754.522} C_VEL
LIN {X 0,Y 404.135,Z 498.146,A -85,B 0,C 180,E1 -10757.295,E2 -10757.295} C_VEL
LIN {X 0,Y 404.157,Z 498.139,A -85,B 0,C 180,E1 -10759.953,E2 -10759.953} C_VEL
LIN {X 0,Y 404.138,Z 498.146,A -85,B 0,C 180,E1 -10763.125,E2 -10763.125} C_VEL
LIN {X 0,Y 404.148,Z 498.14,A -85,B 0,C 180,E1 -10766.187,E2 -10766.187} C_VEL
LIN {X 0,Y 404.149,Z 498.142,A -85,B 0,C 180,E1 -10769.715,E2 -10769.715} C_VEL
LIN {X 0,Y 404.196,Z 498.138,A -85,B 0,C 180,E1 -10773.122,E2 -10773.122} C_VEL
LIN {X 0,Y 404.173,Z 498.142,A -85,B 0,C 180,E1 -10775.334,E2 -10775.334} C_VEL
